(* Logix 5000 project; controller P5 vendor 1 type 14 code 92 rev 20.55; software revision 20.01 *)

TASK MainTask (continuous, watchdog 500 ms) : MainProgram

MODULES
   Local : vendor 1 type 14 code 92 (ICP 0, rev 20.55)
      P5_EN2T_PCN : 1756-EN2T (ICP 1, Ethernet 192.168.1.50, rev 10.1)
         P4 : 1756-EN2T (Ethernet 192.168.1.40, rev 10.1, Output RPI 10 ms)
            P4_CONTROLLER : vendor 1 type 14 code 92 (ICP 0, rev 20.1)
      P5_EN2TR_RIO : vendor 1 type 12 code 200 (ICP 2, Ethernet 192.168.0.40, rev 10.1)
         VSD501 : PowerFlex 525-EENET (Ethernet 192.168.0.57, rev 2.2, Output RPI 20 ms)
         VSD502 : PowerFlex 525-EENET (Ethernet 192.168.0.59, rev 3.1, Output RPI 20 ms)
         RIO5 : 1794-AENTR (Ethernet 192.168.0.52, rev 1.1, Output RPI 20 ms)
            RIO5_DI : 1794-IB32 (Flex 0, rev 1.1, Input RPI 20 ms)
            RIO5_DO : vendor 1 type 7 code 35 (Flex 1, rev 1.1)
            RIO5_AI : 1794-IE12 (Flex 2, rev 1.1, Output RPI 78 ms)
         WRIO5 : vendor 309 type 12 code 1000 (Ethernet 192.168.0.55, rev 3.1, Output RPI 20 ms)
            WRIO5_AI2 : 1734-IE4C (PointIO 2, rev 3.1, Input RPI 80 ms)
            WRIO5_AI1 : vendor 1 type 115 code 210 (PointIO 1, rev 3.1, Input RPI 80 ms)
END_MODULES

TYPE AIN_UDT :
STRUCT
   Pv : REAL;
   Heu : REAL;
   Leu : REAL;
   SAHH : REAL;
   SAH : REAL;
   SAL : REAL;
   SALL : REAL;
   AHH : BOOL;
   AH : BOOL;
   AL : BOOL;
   ALL : BOOL;
   Wifi_Enb : BOOL;
   Hty : BOOL;
   Sim : BOOL;
   Sim_PV : REAL;
END_STRUCT
END_TYPE

TYPE AUTOINP_UDT :
STRUCT
   ON : BOOL;
END_STRUCT
END_TYPE

TYPE ControllerLEDStatus :
STRUCT
   Off : BOOL;
   SolidGreen : BOOL;
   FlashingGreen : BOOL;
   SolidYellow : BOOL;
   FlashingYellow : BOOL;
   FlashingRed : BOOL;
   SolidRed : BOOL;
END_STRUCT
END_TYPE

TYPE DOSING_SETPOINT_UDT :
STRUCT
   High_Setpoint : REAL;
   Low_Setpoint : REAL;
END_STRUCT
END_TYPE

TYPE Duty2_UDT :
STRUCT
   Selection : INT;
   Pump_Running : BOOL;
   Selected_Pmp_Not_Avl : BOOL;
   Both_Pmp_Not_Avl : BOOL;
END_STRUCT
END_TYPE

TYPE FaultRecord :
STRUCT
   timelow : DINT;
   timehigh : DINT;
   type : INT;
   code : INT;
   info : DINT[8];
END_STRUCT
END_TYPE

TYPE FIT_UDT :
STRUCT
   Pv : REAL;
   Heu : REAL;
   Leu : REAL;
   SAHH : REAL;
   SAH : REAL;
   SAL : REAL;
   SALL : REAL;
   Totaliser : REAL;
   AHH : BOOL;
   AH : BOOL;
   AL : BOOL;
   ALL : BOOL;
   Sim : BOOL;
   Sim_PV : REAL;
   Wifi_Enb : BOOL;
   Rst_Totaliser : BOOL;
   Hty : BOOL;
END_STRUCT
END_TYPE

TYPE Logix_Status_FP :
STRUCT
   ClearMinorFaults : DINT;
   Sts_MinorFaultEvents : DINT;
   Sts_MinorFaultBits : DINT;
   Sts_Redundant : DINT;
   Set_FaceplateAnimation : DINT;
   Val_ProductCode : DINT;
   MemoryTemp : INT[29];
   Val_raw_data : INT;
   Sts_IO_LED_raw : INT;
   Sts_ProductCode : INT;
   Val_Force_data_raw : INT;
   MemoryRequestData : SINT[12];
   Sts_Force_Installed : BOOL;
   Sts_Force_Enabled : BOOL;
   Sts_Faulted : BOOL;
   Sts_Run : BOOL;
   Sts_Program : BOOL;
   Sts_Minor_fault : BOOL;
   Sts_Major_fault : BOOL;
   Sts_KS_in_run : BOOL;
   Sts_KS_in_program : BOOL;
   Sts_KS_in_remote : BOOL;
   Sts_Changingmodes : BOOL;
   Sts_Test : BOOL;
   Sts_Ladder_Working : BOOL;
   Cmd_ClearFaultRecord : BOOL;
   Set_Controller_Description : STRING;
   UpdateDelayTimer : TIMER;
   Val_MajorFault : FaultRecord;
   Val_MFS : FaultRecord;
   Sts_IO_LED : ControllerLEDStatus;
   Sts_Battery_LED : ControllerLEDStatus;
   MemoryData : Memory_Data;
   TEST : DINT;
END_STRUCT
END_TYPE

TYPE Memory_Data :
STRUCT
   Free_Mem_IO : DINT;
   Free_Mem_DT : DINT;
   Free_Memory : DINT;
   Total_Mem_IO : DINT;
   Total_Mem_DT : DINT;
   Total_Memory : DINT;
   Biggest_IO_Mem_Size_Ava : DINT;
   Biggest_DT_Mem_Size_Ava : DINT;
END_STRUCT
END_TYPE

TYPE MV_UDT :
STRUCT
   Cmd : INT;
   Status : INT;
   Reset : BOOL;
   Auto : BOOL;
   FTO : BOOL;
   FTC : BOOL;
   Avl : BOOL;
END_STRUCT
END_TYPE

TYPE PLANT_AUTO_UDT :
STRUCT
   ON : BOOL;
   OFF : BOOL;
END_STRUCT
END_TYPE

TYPE PLANT_UDT :
STRUCT
   START : BOOL;
   STOP : BOOL;
END_STRUCT
END_TYPE

TYPE PMP_UDT :
STRUCT
   Cmd : INT;
   Status : INT;
   RunMin : REAL;
   Total_RunMin : REAL;
   RunHr : REAL;
   Total_RunHr : REAL;
   Remote : BOOL;
   Auto : BOOL;
   Fault : BOOL;
   Avl : BOOL;
   Permissive : DINT;
   Shutdown : DINT;
   SD : DINT;
   Reset : BOOL;
   Reset_RunHr : BOOL;
   FTR : BOOL;
   FTS : BOOL;
END_STRUCT
END_TYPE

TYPE PRECONDITION_UDT :
STRUCT
   PERMISSIVE1 : BOOL;
   PERMISSIVE2 : BOOL;
   PERMISSIVE3 : BOOL;
   PERMISSIVE4 : BOOL;
   PERMISSIVE5 : BOOL;
   SHUTDOWN1 : BOOL;
   SHUTDOWN2 : BOOL;
   SHUTDOWN3 : BOOL;
   SHUTDOWN4 : BOOL;
   SHUTDOWN5 : BOOL;
END_STRUCT
END_TYPE

TYPE RED_STAT :
STRUCT
   Redundancy_status_of_the_controller : INT;
   Redundancy_state_of_the_partner : INT;
END_STRUCT
END_TYPE

TYPE SWITCH_UDT :
STRUCT
   Alarm : BOOL;
   Delay : DINT;
END_STRUCT
END_TYPE

TYPE UV_UDT :
STRUCT
   Cmd : INT;
   Status : INT;
   RunMin : REAL;
   Total_RunMin : REAL;
   RunHr : REAL;
   Total_RunHr : REAL;
   Remote : BOOL;
   Auto : BOOL;
   Fault : BOOL;
   Avl : BOOL;
   Permissive : DINT;
   Shutdown : DINT;
   SD : DINT;
   Reset : BOOL;
   Reset_RunHr : BOOL;
   FTR : BOOL;
   FTS : BOOL;
END_STRUCT
END_TYPE

TYPE VSD_UDT :
STRUCT
   Cmd : INT;
   Status : INT;
   RunMin : REAL;
   Total_RunMin : REAL;
   RunHr : REAL;
   Total_RunHr : REAL;
   Remote : BOOL;
   Auto : BOOL;
   Fault : BOOL;
   Avl : BOOL;
   Drive_Ready : BOOL;
   Speed : REAL;
   Speed_Command : REAL;
   Permissive : DINT;
   Shutdown : DINT;
   SD : DINT;
   Reset : BOOL;
   Reset_RunHr : BOOL;
   FTR : BOOL;
   FTS : BOOL;
END_STRUCT
END_TYPE

TYPE WIFI_UDT :
STRUCT
   PLC_WIFI : BOOL;
   RIO_WIFI : BOOL;
END_STRUCT
END_TYPE

ADD_ON_INSTRUCTION AIN_FBD   (* revision 1.0 *)
VAR_INPUT
   WRIO_Enb : BOOL; {visible}
   Raw_RIO : INT; {visible}
   Raw_WRIO : INT; {visible}
   L_Raw_RIO : INT; {visible}
   H_Raw_RIO : INT; {visible}
   L_Raw_WRIO : INT; {visible}
   H_Raw_WRIO : INT; {visible}
   HEU : INT; {visible}
   LEU : INT; {visible}
END_VAR
VAR_OUTPUT
   Hty : BOOL; {visible}
   Wifi_Enb : BOOL; {access Read Only, visible}
   AHH : BOOL; {visible}
   AH : BOOL; {access Read Only, visible}
   AL : BOOL; {access Read Only, visible}
   ALL : BOOL; {visible}
END_VAR
VAR_INPUT
   SAHH : REAL; {visible}
   SAH : REAL; {visible}
   SAL : REAL; {visible}
   SALL : REAL; {visible}
   Simulation : BOOL; {visible}
   RIO_Hty : BOOL; {visible}
   WRIO_Hty : BOOL; {visible}
END_VAR
VAR_IN_OUT
   Pv : REAL; {required}
   Sim_PV : REAL; {required}
   HMI : AIN_UDT; {required}
END_VAR
VAR
   SCALE : SCALE; {access None}
   ALM : ALARM; {access None}
   _Raw : INT; {access None}
   _L_Raw : INT; {access None}
   _H_Raw : INT; {access None}
   _Inst_Hty : BOOL; {access None}
END_VAR

ROUTINE Logic   (* structured text *)
   (*RIO and Wireless RIO Selection*)
   
   IF WRIO_Enb THEN
   	Wifi_Enb	:= 1;
   	_Raw		:= Raw_WRIO;
   	_H_Raw		:= H_Raw_WRIO;
   	_L_Raw		:= L_Raw_WRIO;
   	_Inst_Hty 	:= WRIO_Hty;
   ELSE
   	Wifi_Enb	:= 0;
   	_Raw		:= Raw_RIO;
   	_H_Raw		:= H_Raw_RIO;
   	_L_Raw		:= L_Raw_RIO;
   	_Inst_Hty 	:= RIO_Hty;
   END_IF;
   
   (*Calculation for PV*)
   IF Simulation THEN
   	Pv	:=Sim_PV;
   ELSE
   	SCALE.In		:=_Raw;
   	SCALE.InRawMax	:=_H_Raw;
   	SCALE.InRawMin	:=_L_Raw;
   	SCALE.InEUMax	:=HEU;
   	SCALE.InEUMin	:=LEU;
   	SCL(SCALE);
   
   	IF SCALE.Out<0 THEN
   		Pv	:= 0.0;
   	ELSE
   		Pv	:=SCALE.Out;
   	END_IF;
   
   	Sim_PV	:=Pv;
   
   END_IF;
   
   (*Alarms*)
   ALM.In			:=Pv;
   ALM.HHLimit		:=SAHH;
   ALM.HLimit		:=SAH;
   ALM.LLimit		:=SAL;
   ALM.LLLimit		:=SALL;
   ALM(ALM);
   
   AHH				:=ALM.HHAlarm;
   AH				:=ALM.HAlarm;
   AL				:=ALM.LAlarm;
   ALL				:=ALM.LLAlarm;
   
   Hty:= _Inst_Hty AND (_Raw > _L_Raw) AND (_Raw < _H_Raw)  ;
   
   
   
   
   
   
END_ROUTINE
END_ADD_ON_INSTRUCTION

ADD_ON_INSTRUCTION Duty2_FBD   (* revision 1.0 *)
VAR_INPUT
   AutoInp : BOOL; {visible}
   Selection : INT; {visible}
END_VAR
VAR_OUTPUT
   Start_Pmp1 : BOOL; {visible}
   Start_Pmp2 : BOOL; {visible}
END_VAR
VAR_IN_OUT
   PMP1 : VSD_UDT; {required}
   PMP2 : VSD_UDT; {required}
   HMI : Duty2_UDT; {required}
END_VAR

ROUTINE Logic   (* structured text *)
   IF PMP1.Status=2 OR PMP2.Status=2 THEN
   	HMI.Pump_Running := 1;
   ELSE
   	HMI.Pump_Running := 0;
   END_IF;
   
   HMI.Both_Pmp_Not_Avl		:= NOT PMP1.Avl AND NOT PMP2.Avl;
   
   IF AutoInp THEN
   	CASE Selection OF
   		(*PUMP 1 *)
   		1:
   			IF PMP1.Avl THEN
   				Start_Pmp1					:=1;
   				Start_Pmp2					:=0;
   				HMI.Selected_Pmp_Not_Avl	:=0;
   			ELSIF NOT PMP1.Avl AND PMP2.Avl THEN
   				Start_Pmp1					:=0;
   				Start_Pmp2					:=1;
   				HMI.Selected_Pmp_Not_Avl	:=1;
   			ELSIF NOT PMP1.Avl AND NOT PMP2.Avl	THEN
   				Start_Pmp1					:=0;
   				Start_Pmp2					:=0;
   			ELSE
   				HMI.Selected_Pmp_Not_Avl	:=0;
   			END_IF;
   
   		(*PUMP 2 *)
   		2:
   			IF PMP2.Avl THEN
   				Start_Pmp1					:=0;
   				Start_Pmp2					:=1;
   				HMI.Selected_Pmp_Not_Avl	:=0;
   			ELSIF NOT PMP2.Avl AND PMP1.Avl THEN
   				Start_Pmp1					:=1;
   				Start_Pmp2					:=0;
   				HMI.Selected_Pmp_Not_Avl	:=1;
   			ELSIF NOT PMP1.Avl AND NOT PMP2.Avl	THEN
   				Start_Pmp1					:=0;
   				Start_Pmp2					:=0;
   			ELSE
   				HMI.Selected_Pmp_Not_Avl	:=0;
   			END_IF;
   	END_CASE;
   ELSE
   	Start_Pmp1					:=0;
   	Start_Pmp2					:=0;
   END_IF;
   
   
END_ROUTINE
END_ADD_ON_INSTRUCTION

ADD_ON_INSTRUCTION FIT_FBD   (* revision 1.0 *)
VAR_INPUT
   WRIO_Enb : BOOL; {visible}
   Raw_RIO : INT; {visible}
   Raw_WRIO : INT; {visible}
   L_Raw_RIO : INT; {visible}
   H_Raw_RIO : INT; {visible}
   L_Raw_WRIO : INT; {visible}
   H_Raw_WRIO : INT; {visible}
   HEU : REAL; {visible}
   LEU : REAL; {visible}
END_VAR
VAR_OUTPUT
   Hty : BOOL; {visible}
   Wifi_Enb : BOOL; {visible}
   AHH : BOOL; {visible}
   AH : BOOL; {access Read Only, visible}
   AL : BOOL; {access Read Only, visible}
   ALL : BOOL; {visible}
END_VAR
VAR_INPUT
   SAHH : REAL; {visible}
   SAH : REAL; {visible}
   SAL : REAL; {visible}
   SALL : REAL; {visible}
   Simulation : BOOL; {visible}
   RIO_Hty : BOOL; {visible}
   WRIO_Hty : BOOL; {visible}
   Totaliser_Enb : BOOL; {visible}
   Rst_Totaliser : BOOL; {visible}
END_VAR
VAR_IN_OUT
   Totaliser : REAL; {required}
   Pv : REAL; {required}
   Sim_Pv : REAL; {required}
   HMI : FIT_UDT; {required}
END_VAR
VAR
   SCALE : SCALE; {access None}
   ALM : ALARM; {access None}
   TON : FBD_TIMER; {access None}
   _SEC_P : BOOL; {access None}
   _Inst_Hty : BOOL; {access None}
   _L_Raw : INT; {access None}
   _H_Raw : INT; {access None}
   _Raw : INT; {access None}
   R_TRIG : FBD_ONESHOT; {access None}
END_VAR

ROUTINE Logic   (* structured text *)
   (*RIO and Wireless RIO Selection*)
   
   IF WRIO_Enb THEN
   	Wifi_Enb	:= 1;
   	_Raw		:= Raw_WRIO;
   	_H_Raw		:= H_Raw_WRIO;
   	_L_Raw		:= L_Raw_WRIO;
   	_Inst_Hty 	:= WRIO_Hty;
   ELSE
   	Wifi_Enb	:= 0;
   	_Raw		:= Raw_RIO;
   	_H_Raw		:= H_Raw_RIO;
   	_L_Raw		:= L_Raw_RIO;
   	_Inst_Hty 	:= RIO_Hty;
   END_IF;
   
   (*Calculation for PV*)
   IF Simulation THEN
   	Pv	:= Sim_Pv   ;
   ELSE
   	SCALE.In		:=_Raw;
   	SCALE.InRawMax	:=_H_Raw;
   	SCALE.InRawMin	:=_L_Raw;
   	SCALE.InEUMax	:=HEU;
   	SCALE.InEUMin	:=LEU;
   	SCL(SCALE);
   	IF SCALE.Out>0 THEN
   		Pv	:=SCALE.Out;
   	ELSIF SCALE.Out<=0 THEN
   		Pv	:=0.0;
   	END_IF;
   
   	Sim_Pv	:=Pv;
   END_IF;
   
   (*Alarms*)
   ALM.In			:=Pv;
   ALM.HHLimit		:=SAHH;
   ALM.HLimit		:=SAH;
   ALM.LLimit		:=SAL;
   ALM.LLLimit		:=SALL;
   ALM(ALM);
   
   AHH				:=ALM.HHAlarm;
   AH				:=ALM.HAlarm;
   AL				:=ALM.LAlarm;
   ALL				:=ALM.LLAlarm;
   
   (*SECOND PULSE*)
   TON.PRE	:=1000;
   TON.TimerEnable	:=1;
   TONR(TON );
   R_TRIG.InputBit :=TON.DN ;
   OSRI( R_TRIG);
   _SEC_P  := R_TRIG.OutputBit;
   TON.Reset := _SEC_P;
   
   IF Totaliser_Enb THEN
   	IF _SEC_P THEN
   		HMI.Totaliser := HMI.Totaliser +  (ABS(Pv) / 3600 );
   	END_IF;
   END_IF;
   
   IF  Rst_Totaliser   THEN
   	HMI.Totaliser	:=0;
   END_IF;
   
   Hty:= _Inst_Hty AND (_Raw > _L_Raw) AND (_Raw < _H_Raw)  ;
   
   
   
   
   
   
END_ROUTINE
END_ADD_ON_INSTRUCTION

ADD_ON_INSTRUCTION MV_FBD   (* revision 1.0 *)
VAR_INPUT
   Auto : BOOL; {visible}
END_VAR
VAR_OUTPUT
   Cmd_Open : BOOL; {visible}
   Cmd_Close : BOOL; {visible}
   FTO : BOOL; {visible}
   FTC : BOOL; {access Read Only, visible}
END_VAR
VAR_INPUT
   AutoInp : BOOL; {visible}
   ZSO : BOOL; {visible}
   Open_TM : DINT; {visible}
   ZSC : BOOL; {visible}
   Close_TM : DINT; {visible}
END_VAR
VAR_IN_OUT
   Cmd : INT; {required}
   HMI : MV_UDT; {required}
END_VAR
VAR
   TON_Open_TM : FBD_TIMER; {access None}
   TON_Close_TM : FBD_TIMER; {access None}
END_VAR

ROUTINE Logic   (* structured text *)
   (*Fail to Close*)
   TON_Close_TM.PRE 			:= 	Close_TM*1000;
   TON_Close_TM.TimerEnable 	:=  Cmd_Close;
   TONR(TON_Close_TM);
   
   (*Fail to Open*)
   TON_Open_TM.PRE 			:= 	Open_TM*1000;
   TON_Open_TM.TimerEnable 	:= 	Cmd_Open;
   TONR(TON_Open_TM);
   
   IF ZSC THEN
   	HMI.Status	:=1;
   ELSIF ZSO THEN
   	HMI.Status	:=2;
   ELSE
   	HMI.Status	:=0;
   END_IF;
   
   HMI.Avl:= Auto AND NOT FTC AND NOT FTO;
   
   IF HMI.Reset THEN
   	(*IF NOT TON_Close_TM.DN AND ZSC THEN*)
   			FTC		:= 0;
   	(*END_IF;*)
   	(*IF NOT TON_Open_TM.DN AND ZSO THEN*)
   			FTO		:= 0;
   	(*END_IF;*)
   END_IF;
   
   IF  NOT Auto THEN
   	CASE HMI.Cmd OF
   		1:	(*CLOSE*)
   			Cmd_Close	:= 1;
   			Cmd_Open	:= 0;
   			IF TON_Close_TM.DN AND (NOT ZSC) THEN
   				FTC		:= 1;
   				FTO		:= 0;
   			END_IF;
   		2:	(*OPEN*)
   			IF FTO OR FTC    THEN
   				HMI.Cmd := 1;
   			END_IF;
   
   			IF NOT FTC AND NOT FTO THEN
   				Cmd_Close	:= 0;
   				Cmd_Open	:= 1;
   			END_IF;
   
   			IF TON_Open_TM.DN AND (NOT ZSO) THEN
   				FTC		:= 0;
   				FTO		:= 1;
   				HMI.Cmd := 1;
   			END_IF;
   	END_CASE;
   ELSE
   	(*Maintain Last status when switching from Auto to Manual*)
   	IF ZSO THEN
   		Cmd	:= 2;
   	END_IF;
   	IF ZSC THEN
   		Cmd	:= 1;
   	END_IF;
   
   	IF  AutoInp AND (NOT FTC AND NOT FTO) THEN
   		Cmd_Close	:= 0;
   		Cmd_Open	:= 1;
   		IF TON_Open_TM.DN AND (NOT ZSO) THEN
   			FTC		:= 0;
   			FTO		:= 1;
   		END_IF;
   	ELSE
   		Cmd_Close	:= 1;
   		Cmd_Open	:= 0;
   		IF TON_Close_TM.DN AND (NOT ZSC) THEN
   			FTC		:= 1;
   			FTO		:= 0;
   		END_IF;
   	END_IF;
   END_IF;
   
   
END_ROUTINE
END_ADD_ON_INSTRUCTION

ADD_ON_INSTRUCTION PMP_FBD   (* revision 1.0 *)
VAR_OUTPUT
   Cmd_Start : BOOL; {visible}
   Avl : BOOL; {visible}
   Fault : BOOL; {visible}
   FT_Stop : BOOL; {visible}
   FT_Start : BOOL; {visible}
   RunHr : REAL; {visible}
   Total_RunHr : REAL; {visible}
   SD : DINT; {access Read Only, visible}
END_VAR
VAR_INPUT
   Auto : BOOL; {visible}
   AutoInp : BOOL; {visible}
   Remote : BOOL; {visible}
   Run : BOOL; {visible}
   Trip : BOOL; {visible}
   Start_TM : DINT; {visible}
   Stop_TM : DINT; {visible}
   Rst : BOOL; {visible}
   Rst_RunHr : BOOL; {visible}
   Permissive : DINT; {visible}
   Shutdown : DINT; {visible}
END_VAR
VAR_IN_OUT
   RunMin : REAL; {required}
   Total_RunMin : REAL; {required}
   Cmd : INT; {required}
   HMI : PMP_UDT; {required}
END_VAR
VAR
   TON_Start_TM : FBD_TIMER; {access None}
   TON_Stop_TM : FBD_TIMER; {access None}
   _Min_P : BOOL; {access None}
   TON_Min : FBD_TIMER; {access None}
   R_TRIG_SEC : FBD_ONESHOT; {access None}
END_VAR

ROUTINE Logic   (* structured text *)
   (*Fail to Start*)
   TON_Start_TM.PRE 			:= 	Start_TM*1000;
   TON_Start_TM.TimerEnable 	:=  Cmd_Start;
   TONR(TON_Start_TM);
   
   (*Fail to Stop*)
   TON_Stop_TM.PRE 			:= 	Stop_TM*1000;
   TON_Stop_TM.TimerEnable 	:=  NOT Cmd_Start;
   TONR(TON_Stop_TM);
   
   IF (NOT Run) THEN
   	HMI.Status	:=1;
   ELSE
   	HMI.Status	:=2;
   END_IF;
   
   IF Fault THEN
   	HMI.Fault:= 1;
   ELSE
   	HMI.Fault:= 0;
   END_IF;
   
   IF HMI.Reset THEN
   	IF NOT TON_Stop_TM.DN THEN
   			FT_Stop		:= 0;
   	END_IF;
   	IF NOT TON_Start_TM.DN THEN
   			FT_Start	:= 0;
   	END_IF;
   
   	SD :=0;
   
   END_IF;
   
   Fault		:=Trip OR SD<>0;
   HMI.Remote	:=Remote;
   Avl:= Auto AND Remote AND NOT Fault AND NOT FT_Start AND NOT FT_Stop AND SD=0 ;
   
   IF Remote THEN
   	IF  NOT Auto THEN
   		CASE HMI.Cmd OF
   			1:	(*Stop*)
   				Cmd_Start	:=0;
   				IF TON_Stop_TM.DN AND Run THEN
   					FT_Start	:= 0;
   					FT_Stop		:= 1;
   				END_IF;
   			2:	(*OPEN*)
   				IF NOT Fault AND NOT FT_Start AND NOT FT_Stop AND (Permissive=-1) AND HMI.SD=0 THEN
   					Cmd_Start	:= 1;
   				ELSIF Cmd_Start AND (HMI.SD<>0) OR Fault THEN
   					SD				:= HMI.SD;
   					Cmd_Start		:= 0;
   					HMI.Cmd 		:= 1;
   				ELSIF (Permissive<>-1) THEN
   					HMI.Cmd 		:= 1;
   				END_IF;
   
   				IF TON_Start_TM.DN AND NOT Run THEN
   					FT_Start	:= 1;
   					FT_Stop		:= 0;
   					Cmd_Start	:= 0;
   					HMI.Cmd 	:= 1;
   				END_IF;
   		END_CASE;
   	ELSE
   		IF Run THEN
   			Cmd	:= 2;
   		END_IF;
   		IF (NOT Run) OR Fault OR FT_Start OR FT_Stop THEN
   			Cmd	:= 1;
   		END_IF;
   
   		IF  AutoInp  THEN
   			IF NOT Fault AND NOT FT_Start AND NOT FT_Stop AND (Permissive=-1) AND HMI.SD=0  THEN
   				Cmd_Start	:=1;
   			ELSIF Cmd_Start OR (HMI.SD<>0) OR Fault THEN
   				SD			:= HMI.SD;
   				Cmd_Start	:=0;
   			END_IF;
   
   			IF TON_Start_TM.DN AND NOT Run THEN
   				FT_Start	:= 1;
   				FT_Stop		:= 0;
   				Cmd_Start	:= 0;
   				HMI.Cmd 	:= 1;
   			END_IF;
   		ELSE
   			Cmd_Start	:=0;
   			IF TON_Stop_TM.DN AND Run THEN
   				FT_Start	:= 0;
   				FT_Stop		:= 1;
   
   			END_IF;
   		END_IF;
   	END_IF;
   
   ELSE (*Local*)
   	Cmd_Start	:=0;
   	Cmd	:= 1;
   
   	FT_Start	:= 0;
   	FT_Stop		:= 0;
   
   
   
   
   	(*	IF Run THEN
   			Cmd	:= 2;
   		END_IF;
   		IF (NOT Run) OR Fault OR FT_Start OR FT_Stop THEN
   			Cmd	:= 1;
   		END_IF;
   		*)
   END_IF;
   
   (*1 MIN PULSE*)
   TON_Min.PRE	:=60000;
   TON_Min.TimerEnable	:=1;
   TONR(TON_Min );
   R_TRIG_SEC.InputBit :=TON_Min.DN ;
   OSRI( R_TRIG_SEC);
   _Min_P  := R_TRIG_SEC.OutputBit;
   TON_Min.Reset 	:= _Min_P;
   
   IF Run THEN
   	IF _Min_P THEN
   		RunMin 			:=RunMin + 1.0;
   		Total_RunMin	:=Total_RunMin + 1.0;
   	END_IF;
   END_IF;
   
   RunHr 				:=RunMin/60.0;
   Total_RunHr			:=Total_RunMin/60.0;
   
   IF  Rst_RunHr THEN
   	RunMin	:=0;
   END_IF;
   
   
   
END_ROUTINE
END_ADD_ON_INSTRUCTION

ADD_ON_INSTRUCTION SWITCH_FBD   (* revision 1.0 *)
VAR_INPUT
   Alarm : BOOL; {visible}
   Delay : DINT; {required}
END_VAR
VAR_OUTPUT
   Status : BOOL; {access None, required}
END_VAR
VAR_IN_OUT
   HMI : SWITCH_UDT; {required}
END_VAR
VAR
   TON_Delay_Sec : FBD_TIMER; {access None}
END_VAR

ROUTINE Logic   (* structured text *)
   (*Delay for Alarm*)
   TON_Delay_Sec.PRE 			:= 	Delay*1000;
   TON_Delay_Sec.TimerEnable 	:=  Alarm;
   TONR(TON_Delay_Sec);
   
   Status := TON_Delay_Sec.DN ;
END_ROUTINE
END_ADD_ON_INSTRUCTION

ADD_ON_INSTRUCTION UV_FBD   (* revision 1.0 *)
VAR_OUTPUT
   Cmd_Start : BOOL; {visible}
   Avl : BOOL; {visible}
   Fault : BOOL; {visible}
   FT_Stop : BOOL; {visible}
   FT_Start : BOOL; {visible}
   RunHr : REAL; {visible}
   Total_RunHr : REAL; {visible}
END_VAR
VAR_INPUT
   Auto : BOOL; {visible}
   AutoInp : BOOL; {visible}
   Remote : BOOL; {visible}
   Run : BOOL; {visible}
   Trip : BOOL; {visible}
   Start_TM : DINT; {visible}
   Stop_TM : DINT; {visible}
   Rst : BOOL; {visible}
   Rst_RunHr : BOOL; {visible}
   Permissive : INT; {visible}
   Shutdown : INT; {visible}
END_VAR
VAR_IN_OUT
   RunMin : REAL; {required}
   Total_RunMin : REAL; {required}
   Cmd : INT; {required}
   HMI : UV_UDT; {required}
END_VAR
VAR
   TON_Start_TM : FBD_TIMER; {access None}
   TON_Stop_TM : FBD_TIMER; {access None}
   _Min_P : BOOL; {access None}
   TON_Min : FBD_TIMER; {access None}
   R_TRIG_SEC : FBD_ONESHOT; {access None}
END_VAR

ROUTINE Logic   (* structured text *)
   (*Fail to Start*)
   TON_Start_TM.PRE 			:= 	Start_TM*1000;
   TON_Start_TM.TimerEnable 	:=  Cmd_Start;
   TONR(TON_Start_TM);
   
   (*Fail to Stop*)
   TON_Stop_TM.PRE 			:= 	Stop_TM*1000;
   TON_Stop_TM.TimerEnable 	:=  NOT Cmd_Start;
   TONR(TON_Stop_TM);
   
   IF (NOT Run) THEN
   	HMI.Status	:=1;
   ELSE
   	HMI.Status	:=2;
   END_IF;
   
   IF Fault THEN
   	HMI.Fault:= 1;
   ELSE
   	HMI.Fault:= 0;
   END_IF;
   
   IF HMI.Reset THEN
   	IF NOT TON_Stop_TM.DN THEN
   			FT_Stop		:= 0;
   	END_IF;
   	IF NOT TON_Start_TM.DN THEN
   			FT_Start	:= 0;
   	END_IF;
   END_IF;
   
   
   HMI.Remote	:=Remote;
   Avl:= Auto AND Remote AND NOT Fault AND NOT FT_Stop AND NOT FT_Stop   ;
   
   
   
   IF Remote THEN
   	IF  NOT Auto THEN
   		CASE HMI.Cmd OF
   			1:	(*Stop*)
   				Cmd_Start	:=0;
   				IF TON_Stop_TM.DN AND Run THEN
   					FT_Start	:= 0;
   					FT_Stop		:= 1;
   				END_IF;
   			2:	(*OPEN*)
   				IF NOT Fault AND (NOT FT_Start OR FT_Stop) AND (Permissive=-1) THEN
   					Cmd_Start	:= 1;
   				END_IF;
   
   				IF (Shutdown<>0) OR Fault THEN
   					Cmd_Start	:= 0;
   					HMI.Cmd 	:= 1;
   				END_IF;
   
   				IF TON_Start_TM.DN AND NOT Run THEN
   					FT_Start	:= 1;
   					FT_Stop		:= 0;
   					Cmd_Start	:= 0;
   					HMI.Cmd 	:= 1;
   				END_IF;
   		END_CASE;
   	ELSE
   		IF Run THEN
   			Cmd	:= 2;
   		END_IF;
   		IF (NOT Run) OR Fault OR FT_Start OR FT_Stop THEN
   			Cmd	:= 1;
   		END_IF;
   
   		IF  AutoInp  THEN
   			IF NOT Fault AND (NOT FT_Start OR FT_Stop) AND (Permissive=-1) THEN
   				Cmd_Start	:=1;
   			END_IF;
   
   			IF (Shutdown<>0) OR Fault THEN
   				Cmd_Start	:=0;
   			END_IF;
   
   			IF TON_Start_TM.DN AND NOT Run THEN
   				FT_Start	:= 1;
   				FT_Stop		:= 0;
   				Cmd_Start	:= 0;
   				HMI.Cmd 	:= 1;
   			END_IF;
   		ELSE
   			Cmd_Start	:=0;
   			IF TON_Stop_TM.DN AND Run THEN
   				FT_Start	:= 0;
   				FT_Stop		:= 1;
   
   			END_IF;
   		END_IF;
   	END_IF;
   
   ELSE (*Local*)
   	Cmd_Start	:=0;
   	Cmd	:= 1;
   
   	(*	IF Run THEN
   			Cmd	:= 2;
   		END_IF;
   		IF (NOT Run) OR Fault OR FT_Start OR FT_Stop THEN
   			Cmd	:= 1;
   		END_IF;
   		*)
   END_IF;
   
   (*1 MIN PULSE*)
   TON_Min.PRE	:=60000;
   TON_Min.TimerEnable	:=1;
   TONR(TON_Min );
   R_TRIG_SEC.InputBit :=TON_Min.DN ;
   OSRI( R_TRIG_SEC);
   _Min_P  := R_TRIG_SEC.OutputBit;
   TON_Min.Reset 	:= _Min_P;
   
   IF Run THEN
   	IF _Min_P THEN
   		RunMin 			:=RunMin + 1.0;
   		Total_RunMin	:=Total_RunMin + 1.0;
   	END_IF;
   END_IF;
   
   RunHr 				:=RunMin/60.0;
   Total_RunHr			:=Total_RunMin/60.0;
   
   IF  Rst_RunHr THEN
   	RunMin	:=0;
   END_IF;
   
   
   
END_ROUTINE
END_ADD_ON_INSTRUCTION

ADD_ON_INSTRUCTION VSD_FBD   (* revision 1.0 *)
VAR_OUTPUT
   Avl : BOOL; {visible}
   Fault : BOOL; {visible}
   FT_Stop : BOOL; {visible}
   FT_Start : BOOL; {visible}
   RunHr : REAL; {visible}
   Total_RunHr : REAL; {visible}
   Speed : REAL; {visible}
   Rdy : BOOL; {visible}
   SD : DINT; {access Read Only, visible}
END_VAR
VAR_INPUT
   Auto : BOOL; {visible}
   AutoInp : BOOL; {visible}
   Remote : BOOL; {visible}
   Run : BOOL; {visible}
   Trip : BOOL; {visible}
   Start_PB : BOOL; {visible}
   Start_TM : DINT; {visible}
   Stop_TM : DINT; {visible}
   Rst : BOOL; {visible}
   Rst_RunHr : BOOL; {visible}
   AutoSpeed : REAL; {visible}
   Speed_Cmd : REAL; {visible}
   Permissive : DINT; {visible}
   Shutdown : DINT; {visible}
END_VAR
VAR_IN_OUT
   VSD_In : AB:PowerFlex525V_EENET_Drive:I:0; {required}
   VSD_Out : AB:PowerFlex525V_EENET_Drive:O:0; {required}
   RunMin : REAL; {required}
   Total_RunMin : REAL; {required}
   Cmd : INT; {required}
   HMI : VSD_UDT; {required}
END_VAR
VAR
   TON_Start_TM : FBD_TIMER; {access None}
   TON_Stop_TM : FBD_TIMER; {access None}
   _Min_P : BOOL; {access None}
   TON_Min : FBD_TIMER; {access None}
   R_TRIG_SEC : FBD_ONESHOT; {access None}
END_VAR

ROUTINE Logic   (* structured text *)
   (*Fail to Start*)
   TON_Start_TM.PRE 			:= 	Start_TM*1000;
   TON_Start_TM.TimerEnable 	:=  VSD_Out.Start;
   TONR(TON_Start_TM);
   
   (*Fail to Stop*)
   TON_Stop_TM.PRE 			:= 	Stop_TM*1000;
   TON_Stop_TM.TimerEnable 	:=  VSD_Out.Stop;
   TONR(TON_Stop_TM);
   
   IF (NOT VSD_In.Active) THEN
   	HMI.Status	:=1;
   ELSE
   	HMI.Status	:=2;
   END_IF;
   
   Rdy				:= VSD_In.Ready;
   Speed			:= VSD_In.OutputFreq/100;
   HMI.Remote		:= Remote;
   
   Avl:= Auto AND Remote AND NOT Fault AND NOT FT_Start AND NOT FT_Stop AND SD=0;  ;
   HMI.Fault:= VSD_In.Faulted OR Trip OR SD<>0;
   
   
   
   IF HMI.Reset THEN
   	VSD_Out.ClearFaults:=1;
   	HMI.SHUTDOWN:=0;
   
   	IF NOT TON_Stop_TM.DN THEN
   			FT_Stop		:= 0;
   	END_IF;
   	IF NOT TON_Start_TM.DN THEN
   			FT_Start	:= 0;
   	END_IF;
   
   	SD:=0;
   END_IF;
   
   IF Remote THEN
   	IF  NOT Auto THEN
   		CASE HMI.Cmd OF
   			1:	(*Stop*)
   
   				VSD_Out.Start		:=0;
   				VSD_Out.Stop		:=1;
   				VSD_Out.FreqCommand	:=Speed_Cmd;
   
   				IF TON_Stop_TM.DN AND VSD_In.Active THEN
   					FT_Start	:= 0;
   					FT_Stop		:= 1;
   				END_IF;
   			2:	(*Start*)
   				IF NOT VSD_In.Faulted AND (NOT FT_Start OR FT_Stop) AND (Permissive=-1) AND HMI.SD=0 THEN
   					VSD_Out.Start		:=1;
   					VSD_Out.Stop		:=0;
   			        VSD_Out.FreqCommand	:=Speed_Cmd*100;
   
   				ELSIF VSD_Out.Start OR (HMI.SD<>0) OR Fault THEN
   					SD 					:=HMI.SD;
   					VSD_Out.Start		:=0;
   					VSD_Out.Stop		:=1;
   					VSD_Out.FreqCommand	:=Speed_Cmd*100;
   					HMI.Cmd 	:= 1;
   				ELSIF (Permissive<>-1) THEN
   					HMI.Cmd 		:= 1;
   				END_IF;
   
   				IF TON_Start_TM.DN AND NOT Run THEN
   					FT_Start		:=1;
   					FT_Stop			:=0;
   					VSD_Out.Start	:=0;
   					VSD_Out.Stop	:=1;
   					HMI.Cmd 		:=1;
   				END_IF;
   		END_CASE;
   	ELSE
   		IF VSD_In.Active THEN
   			Cmd	:= 2;
   		END_IF;
   		IF (NOT VSD_In.Active) OR VSD_In.Faulted OR FT_Start OR FT_Stop THEN
   			Cmd	:= 1;
   		END_IF;
   
   		IF  AutoInp  THEN
   			IF NOT VSD_In.Faulted AND (NOT FT_Start OR FT_Stop) AND (Permissive=-1) AND HMI.SD=0 THEN
   				VSD_Out.Start		:=1;
   				VSD_Out.Stop		:=0;
   				VSD_Out.FreqCommand	:=AutoSpeed*100;
   
   			ELSIF VSD_Out.Start OR (HMI.SD<>0) OR Fault THEN
   				SD 					:=HMI.SD;
   				VSD_Out.Start		:=0;
   				VSD_Out.Stop		:=1;
   				VSD_Out.FreqCommand	:=AutoSpeed*100;
   				HMI.Cmd 			:= 1;
   			END_IF;
   
   			IF TON_Start_TM.DN AND NOT VSD_In.Active THEN
   				VSD_Out.Start		:=0;
   				VSD_Out.Stop		:=1;
   				VSD_Out.FreqCommand	:=AutoSpeed*100;
   				HMI.Cmd 			:= 1;
   			END_IF;
   		ELSE
   				VSD_Out.Start		:=0;
   				VSD_Out.Stop		:=1;
   			IF TON_Stop_TM.DN AND VSD_In.Active THEN
   				FT_Start	:= 0;
   				FT_Stop		:= 1;
   
   			END_IF;
   		END_IF;
   	END_IF;
   
   ELSE (*Local*)
   		IF Start_PB THEN
   			VSD_Out.Start 	:=1;
   			VSD_Out.Stop	:=0;
   				(*	VSD_Out.FreqCommand	:=Speed_Cmd*100; *)
   				 VSD_Out.FreqCommand	:=Speed_Cmd*110;
   		ELSE
   			VSD_Out.Start 	:=0;
   			VSD_Out.Stop	:=1;
   				(*	VSD_Out.FreqCommand	:=Speed_Cmd*100; *)
   				 VSD_Out.FreqCommand	:=Speed_Cmd*110;
   		END_IF;
   
   
   		IF Run THEN
   			Cmd	:= 2;
   		END_IF;
   		IF (NOT Run) OR Fault OR FT_Start OR FT_Stop THEN
   			Cmd	:= 1;
   		END_IF;
   END_IF;
   
   (*1 MIN PULSE*)
   TON_Min.PRE	:=60000;
   TON_Min.TimerEnable	:=1;
   TONR(TON_Min );
   R_TRIG_SEC.InputBit :=TON_Min.DN ;
   OSRI( R_TRIG_SEC);
   _Min_P  := R_TRIG_SEC.OutputBit;
   TON_Min.Reset 	:= _Min_P;
   
   IF Run OR VSD_In.Active THEN
   	IF _Min_P THEN
   		RunMin :=RunMin + 1.0;
   		Total_RunMin	:=Total_RunMin + 1.0;
   	END_IF;
   END_IF;
   
   RunHr 				:=RunMin/60.0;
   Total_RunHr			:=Total_RunMin/60.0;
   
   IF  Rst_RunHr THEN
   	RunMin	:=0;
   END_IF;
   
   
   
END_ROUTINE
END_ADD_ON_INSTRUCTION

VAR_GLOBAL   (* controller tags *)
   _FIT501_Tot_Enb : BOOL;
   _FIT502_Tot_Enb : BOOL;
   _FIT503_Tot_Enb : BOOL := 1;
   _FIT504_Tot_Enb : BOOL := 1;
   _MIN_P : BOOL;
   _MV501_AutoInp : BOOL;
   _MV502_AutoInp : BOOL;
   _MV503_AutoInp : BOOL;
   _MV504_AutoInp : BOOL;
   _NEXT : BOOL;
   _P401_AutoInp : BOOL;
   _P402_AutoInp : BOOL;
   _P403_AutoInp : BOOL;
   _P404_AutoInp : BOOL;
   _P501_AutoInp : BOOL;
   _P501_AutoSpeed : REAL;
   _P502_AutoInp : BOOL;
   _P502_AutoSpeed : REAL;
   _P50X_AutoSpeed : REAL := 10.0;
   _P_NAHSO3_ORP_DUTY_AutoInp : BOOL;
   _P_NAHSO3_ORP_DUTY_SR : DOMINANT_SET := (Reset := 1, OutNot := 1);
   _P_RO_FEED_DUTY_AutoInp : BOOL;
   _P_RO_FEED_DUTY_SR : DOMINANT_SET := (Set := 1, Out := 1);
   _P_RO_HIGH_AutoInp : BOOL;
   _P_UF_FEED_DUTY_AutoInp : BOOL := 1;
   _SEC_P : BOOL;
   _SEC_P1 : BOOL;
   _SEC_TEST : INT := -6124;
   _SEC_TEST1 : INT := 2391;
   _STOP : BOOL;
   _UV401_AutoInp : BOOL := 1;
   _UV_SR : DOMINANT_SET := (Set := 1, Out := 1);
   AI_AIT_401_HRDNSS : INT := -11;
   AI_AIT_401_HRDNSS_HTY : BOOL := 1;
   AI_AIT_402_ORP : INT := -17;
   AI_AIT_402_ORP_HTY : BOOL := 1;
   AI_AIT_501_PH : INT := 18894;
   AI_AIT_501_PH_HTY : BOOL := 1;
   AI_AIT_502_ORP : INT := 9002;
   AI_AIT_502_ORP_HTY : BOOL := 1;
   AI_AIT_503_COND : INT := 5384;
   AI_AIT_503_COND_HTY : BOOL := 1;
   AI_AIT_504_COND : INT := 933;
   AI_AIT_504_COND_HTY : BOOL := 1;
   AI_FIT_401_FLOW : INT := -19;
   AI_FIT_401_FLOW_HTY : BOOL := 1;
   AI_FIT_501_FLOW : INT := 15;
   AI_FIT_501_FLOW_HTY : BOOL := 1;
   AI_FIT_502_FLOW : INT := -9;
   AI_FIT_502_FLOW_HTY : BOOL := 1;
   AI_FIT_503_FLOW : INT := -24;
   AI_FIT_503_FLOW_HTY : BOOL := 1;
   AI_FIT_504_FLOW : INT := -26;
   AI_FIT_504_FLOW_HTY : BOOL := 1;
   AI_LIT_401_LEVEL : INT := -9;
   AI_LIT_401_LEVEL_HTY : BOOL := 1;
   AI_PIT_501_PRESS : INT := 722;
   AI_PIT_501_PRESS_HTY : BOOL := 1;
   AI_PIT_502_PRESS : INT := -21;
   AI_PIT_502_PRESS_HTY : BOOL := 1;
   AI_PIT_503_PRESS : INT := 402;
   AI_PIT_503_PRESS_HTY : BOOL := 1;
   AI_RIO4_SPARE_03 : INT;
   AI_RIO4_SPARE_03_HTY : BOOL;
   AI_RIO4_SPARE_04 : INT;
   AI_RIO4_SPARE_04_HTY : BOOL;
   AI_RIO4_SPARE_05 : INT;
   AI_RIO4_SPARE_05_HTY : BOOL;
   AI_RIO4_SPARE_06 : INT;
   AI_RIO4_SPARE_06_HTY : BOOL;
   AI_RIO4_SPARE_07 : INT;
   AI_RIO4_SPARE_07_HTY : BOOL;
   AI_RIO4_SPARE_08 : INT;
   AI_RIO4_SPARE_08_HTY : BOOL;
   AI_RIO4_SPARE_09 : INT;
   AI_RIO4_SPARE_09_HTY : BOOL;
   AI_RIO4_SPARE_10 : INT;
   AI_RIO4_SPARE_10_HTY : BOOL;
   AI_RIO4_SPARE_11 : INT;
   AI_RIO4_SPARE_11_HTY : BOOL := 1;
   AI_RIO5_SPARE_11 : INT := -7703;
   AIT401_FB : AIN_FBD := (Raw_RIO := -11, Raw_WRIO := 3266, H_Raw_RIO := 31208, L_Raw_WRIO := 3277, H_Raw_WRIO := 16383, HEU := 2, Hty := 1, AL := 1, ALL := 1, RIO_Hty := 1);
   AIT401_FB_01 : AIN_FBD;
   AIT402_FB : AIN_FBD := (Raw_RIO := -17, Raw_WRIO := 3268, H_Raw_RIO := 31208, L_Raw_WRIO := 3277, H_Raw_WRIO := 16383, HEU := 2, Hty := 1, AL := 1, ALL := 1, RIO_Hty := 1);
   AIT501_FB : AIN_FBD := (Raw_RIO := 18889, Raw_WRIO := 10247, H_Raw_RIO := 31208, L_Raw_WRIO := 3277, H_Raw_WRIO := 16383, HEU := 12, LEU := 2, Hty := 1, AHH := 1, AH := 1, RIO_Hty := 1);
   AIT502_FB : AIN_FBD := (Raw_RIO := 9002, Raw_WRIO := 6637, H_Raw_RIO := 31208, L_Raw_WRIO := 3277, H_Raw_WRIO := 16383, HEU := 800, Hty := 1, SAHH := 300.0, SAH := 250.0, RIO_Hty := 1);
   AIT503_FB : AIN_FBD := (Raw_RIO := 5384, Raw_WRIO := 6434, H_Raw_RIO := 31208, L_Raw_WRIO := 3277, H_Raw_WRIO := 16383, HEU := 1000, Hty := 1, AL := 1, SAHH := 500.0, SAH := 260.0, SAL := 250.0, RIO_Hty := 1);
   AIT504_FB : AIN_FBD := (Raw_RIO := 944, Raw_WRIO := 3355, H_Raw_RIO := 31208, L_Raw_WRIO := 3277, H_Raw_WRIO := 16383, HEU := 1200, Hty := 1, SAHH := 50.0, SAH := 40.0, RIO_Hty := 1);
   DI_DPSH_301_HIGH : BOOL;
   DI_LS_401_LOW : BOOL;
   DI_MV_501_ZSC : BOOL := 1;
   DI_MV_501_ZSO : BOOL;
   DI_MV_502_ZSC : BOOL := 1;
   DI_MV_502_ZSO : BOOL;
   DI_MV_503_ZSC : BOOL := 1;
   DI_MV_503_ZSO : BOOL;
   DI_MV_504_ZSC : BOOL := 1;
   DI_MV_504_ZSO : BOOL;
   DI_P_401_AUTO : BOOL := 1;
   DI_P_401_FAULT : BOOL;
   DI_P_401_RUN : BOOL;
   DI_P_402_AUTO : BOOL := 1;
   DI_P_402_FAULT : BOOL;
   DI_P_402_RUN : BOOL;
   DI_P_403_AUTO : BOOL := 1;
   DI_P_403_FAULT : BOOL;
   DI_P_403_RUN : BOOL;
   DI_P_404_AUTO : BOOL := 1;
   DI_P_404_FAULT : BOOL;
   DI_P_404_RUN : BOOL;
   DI_P_501_AUTO : BOOL := 1;
   DI_P_501_FAULT : BOOL;
   DI_P_501_RUN : BOOL;
   DI_P_502_AUTO : BOOL := 1;
   DI_P_502_FAULT : BOOL;
   DI_P_502_RUN : BOOL;
   DI_PSH_501_HIGH : BOOL;
   DI_PSL_501_LOW : BOOL;
   DI_RIO4_SPARE_10 : BOOL;
   DI_RIO4_SPARE_11 : BOOL;
   DI_RIO4_SPARE_12 : BOOL;
   DI_RIO4_SPARE_13 : BOOL;
   DI_RIO4_SPARE_14 : BOOL;
   DI_RIO4_SPARE_15 : BOOL;
   DI_RIO4_SPARE_16 : BOOL;
   DI_RIO4_SPARE_17 : BOOL;
   DI_RIO4_SPARE_19 : BOOL;
   DI_RIO4_SPARE_20 : BOOL;
   DI_RIO4_SPARE_21 : BOOL;
   DI_RIO4_SPARE_22 : BOOL;
   DI_RIO4_SPARE_23 : BOOL;
   DI_RIO4_SPARE_24 : BOOL;
   DI_RIO4_SPARE_25 : BOOL;
   DI_RIO4_SPARE_26 : BOOL;
   DI_RIO4_SPARE_27 : BOOL;
   DI_RIO4_SPARE_28 : BOOL;
   DI_RIO4_SPARE_29 : BOOL;
   DI_RIO4_SPARE_30 : BOOL;
   DI_RIO4_SPARE_31 : BOOL;
   DI_RIO5_SPARE_19 : BOOL;
   DI_RIO5_SPARE_20 : BOOL;
   DI_RIO5_SPARE_21 : BOOL;
   DI_RIO5_SPARE_22 : BOOL;
   DI_RIO5_SPARE_23 : BOOL;
   DI_RIO5_SPARE_24 : BOOL;
   DI_RIO5_SPARE_25 : BOOL;
   DI_RIO5_SPARE_26 : BOOL;
   DI_RIO5_SPARE_27 : BOOL;
   DI_RIO5_SPARE_28 : BOOL;
   DI_RIO5_SPARE_29 : BOOL;
   DI_RIO5_SPARE_30 : BOOL;
   DI_RIO5_SPARE_31 : BOOL;
   DI_UV_401_AUTO : BOOL := 1;
   DI_UV_401_FAULT : BOOL;
   DI_UV_401_RUN : BOOL;
   DI_UV_402_FAULT : BOOL;
   DI_UV_402_RUN : BOOL;
   DI_VSD_1_PB : BOOL;
   DI_VSD_2_PB : BOOL;
   DI_WIFI_PLC_4 : BOOL := 1;
   DI_WIFI_PLC_5 : BOOL;
   DI_WIFI_RIO_4 : BOOL;
   DI_WIFI_RIO_5 : BOOL;
   DO_MV_501_CLOSE : BOOL := 1;
   DO_MV_501_OPEN : BOOL;
   DO_MV_502_CLOSE : BOOL := 1;
   DO_MV_502_OPEN : BOOL;
   DO_MV_503_CLOSE : BOOL := 1;
   DO_MV_503_OPEN : BOOL;
   DO_MV_504_CLOSE : BOOL := 1;
   DO_MV_504_OPEN : BOOL;
   DO_P_401_START : BOOL;
   DO_P_402_START : BOOL;
   DO_P_403_START : BOOL;
   DO_P_404_START : BOOL;
   DO_RIO4_SPARE_04 : BOOL;
   DO_RIO4_SPARE_05 : BOOL;
   DO_RIO4_SPARE_06 : BOOL;
   DO_RIO4_SPARE_07 : BOOL;
   DO_RIO4_SPARE_08 : BOOL;
   DO_RIO4_SPARE_09 : BOOL;
   DO_RIO4_SPARE_10 : BOOL;
   DO_RIO4_SPARE_11 : BOOL;
   DO_RIO4_SPARE_12 : BOOL;
   DO_RIO4_SPARE_13 : BOOL;
   DO_RIO4_SPARE_14 : BOOL;
   DO_RIO4_SPARE_15 : BOOL;
   DO_RIO5_SPARE_04 : BOOL;
   DO_RIO5_SPARE_05 : BOOL;
   DO_RIO5_SPARE_06 : BOOL;
   DO_RIO5_SPARE_07 : BOOL;
   DO_RIO5_SPARE_08 : BOOL;
   DO_RIO5_SPARE_09 : BOOL;
   DO_RIO5_SPARE_10 : BOOL;
   DO_RIO5_SPARE_11 : BOOL;
   DO_RIO5_SPARE_12 : BOOL;
   DO_RIO5_SPARE_13 : BOOL;
   DO_RIO5_SPARE_14 : BOOL;
   DO_RIO5_SPARE_15 : BOOL;
   DO_UV_401_START : BOOL;
   DUMMY_AIT : AIN_UDT;
   FIT401_FB : FIT_FBD := (Raw_RIO := -19, Raw_WRIO := 3263, L_Raw_RIO := 6242, H_Raw_RIO := 31208, L_Raw_WRIO := 3277, H_Raw_WRIO := 16383, HEU := 5.0, Hty := 1, AL := 1, ALL := 1, RIO_Hty := 1);
   FIT501_FB : FIT_FBD := (Raw_RIO := 15, Raw_WRIO := 8777, H_Raw_RIO := 31208, L_Raw_WRIO := 3277, H_Raw_WRIO := 16383, HEU := 4.0, Hty := 1, AL := 1, SAHH := 3.0, SAH := 2.0, SAL := 1.0, RIO_Hty := 1);
   FIT502_FB : FIT_FBD := (Raw_RIO := -9, Raw_WRIO := 7239, L_Raw_RIO := -20, H_Raw_RIO := 31208, L_Raw_WRIO := 3277, H_Raw_WRIO := 16383, HEU := 4.0, Hty := 1, AHH := 1, AH := 1, RIO_Hty := 1);
   FIT503_FB : FIT_FBD := (Raw_RIO := -24, Raw_WRIO := 5689, L_Raw_RIO := -35, H_Raw_RIO := 31208, L_Raw_WRIO := 3277, H_Raw_WRIO := 16383, HEU := 4.0, Hty := 1, AHH := 1, AH := 1, RIO_Hty := 1, Totaliser_Enb := 1);
   FIT504_FB : FIT_FBD := (Raw_RIO := -26, Raw_WRIO := 5188, L_Raw_RIO := -15, H_Raw_RIO := 31208, L_Raw_WRIO := 3277, H_Raw_WRIO := 16383, HEU := 2.0, AL := 1, ALL := 1, SAHH := 3.5, SAH := 1.0, RIO_Hty := 1, Totaliser_Enb := 1);
   HMI_AIT401 : AIN_UDT := (Pv := -0.00070494745, AL := 1, ALL := 1, Hty := 1);
   HMI_AIT402 : AIN_UDT := (Pv := -0.0010894643, AL := 1, ALL := 1, Hty := 1);
   HMI_AIT501 : AIN_UDT := (Pv := 8.054216, AHH := 1, AH := 1, Hty := 1, Sim_PV := 8.054216);
   HMI_AIT502 : AIN_UDT := (Pv := 230.91515, SAHH := 300.0, SAH := 250.0, Hty := 1, Sim_PV := 230.91515);
   HMI_AIT503 : AIN_UDT := (Pv := 172.51987, SAHH := 500.0, SAH := 260.0, SAL := 250.0, AL := 1, Hty := 1, Sim_PV := 172.51987);
   HMI_AIT504 : AIN_UDT := (Pv := 36.298386, SAHH := 50.0, SAH := 40.0, Hty := 1, Sim_PV := 36.298386);
   HMI_FIT401 : FIT_UDT := (Pv := 0.0010243934, SAHH := 3.0, SAH := 2.0, SAL := 0.5, SALL := 0.4, Totaliser := 381.51465, AL := 1, ALL := 1, Sim_PV := 0.0010243934, Hty := 1);
   HMI_FIT501 : FIT_UDT := (Pv := 0.001922584, SAHH := 3.0, SAH := 2.0, SAL := 1.0, Totaliser := 448.75452, AL := 1, Sim_PV := 0.001922584, Hty := 1);
   HMI_FIT502 : FIT_UDT := (Pv := 0.001408992, Totaliser := 331.85107, AHH := 1, AH := 1, Sim_PV := 0.001408992, Hty := 1);
   HMI_FIT503 : FIT_UDT := (Pv := 0.0014083155, Totaliser := 52.980667, AHH := 1, AH := 1, Sim_PV := 0.0014083155, Hty := 1);
   HMI_FIT504 : FIT_UDT := (SAHH := 3.5, SAH := 1.0, Totaliser := 129.2501, AL := 1, ALL := 1);
   HMI_FLUSHING_MIN : INT;
   HMI_FLUSHING_MIN_SP : INT := 1;
   HMI_HIGH_RO_MAX_SPEED : REAL;
   HMI_HIGH_RO_MIN_SPEED : REAL := 10.0;
   HMI_HPP_Q_MAX_M3H : REAL := 2.0;
   HMI_HPP_Q_SET_M3H : REAL := 1.25;
   HMI_LIT401 : AIN_UDT := (Pv := -0.0005767752, AL := 1, ALL := 1, Hty := 1);
   HMI_LS401 : SWITCH_UDT;
   HMI_MIN_RO_VSD_SPEED : REAL := 3.125;
   HMI_MV501 : MV_UDT := (Cmd := 1, Status := 1, Reset := 1, Auto := 1, Avl := 1);
   HMI_MV501_TIMEOUT_TM : INT;
   HMI_MV502 : MV_UDT := (Cmd := 1, Status := 1, Reset := 1, Auto := 1, Avl := 1);
   HMI_MV502_TIMEOUT_TM : INT;
   HMI_MV503 : MV_UDT := (Cmd := 1, Status := 1, Reset := 1, Auto := 1, Avl := 1);
   HMI_MV503_TIMEOUT_TM : INT;
   HMI_MV504 : MV_UDT := (Cmd := 1, Status := 1, Reset := 1, Auto := 1, Avl := 1);
   HMI_MV504_TIMEOUT_TM : INT;
   HMI_NAHSO3_ORP_DOSING : DOSING_SETPOINT_UDT;
   HMI_P401 : PMP_UDT := (Status := 2, Remote := 1, Permissive := -1);
   HMI_P402 : PMP_UDT := (Status := 1, Remote := 1, Permissive := -1);
   HMI_P403 : PMP_UDT := (Status := 1, Remote := 1, Permissive := -1);
   HMI_P404 : PMP_UDT := (Status := 1, Remote := 1, Permissive := -1);
   HMI_P4_PERMISSIVE : BOOL;
   HMI_P4_STATE : INT;
   HMI_P501 : VSD_UDT := (Cmd := 1, Status := 1, Total_RunMin := 17445.0, Total_RunHr := 290.75, Remote := 1, Auto := 1, Avl := 1, Speed_Command := 10.0, Permissive := -2, SD := 1, Reset := 1, Reset_RunHr := 1);
   HMI_P501_MSG : PRECONDITION_UDT := (PERMISSIVE2 := 1, PERMISSIVE3 := 1);
   HMI_P502 : VSD_UDT := (Cmd := 1, Status := 1, RunMin := 409.0, Total_RunMin := 409.0, RunHr := 6.8166666, Total_RunHr := 6.8166666, Remote := 1, Auto := 1, Avl := 1, Drive_Ready := 1, Speed_Command := 35.0, Permissive := -8, SD := 5, Reset := 1);
   HMI_P502_MSG : PRECONDITION_UDT;
   HMI_P5_PERMISSIVE : AUTOINP_UDT := (ON := 1);
   HMI_P5_SD_FLUSHING_DONE : AUTOINP_UDT;
   HMI_P5_STATE : INT := 1;
   HMI_P_NAHSO3_ORP_DUTY : Duty2_UDT;
   HMI_P_RO_FEED_DUTY : Duty2_UDT := (Selection := 1);
   HMI_P_RO_HIGH_DUTY : Duty2_UDT := (Selection := 1);
   HMI_P_UF_FEED_DUTY : Duty2_UDT;
   HMI_PERMEATE_COND_SP : REAL := 300.0;
   HMI_PERMEATE_FLOW_SP : REAL;
   HMI_PIT501 : AIN_UDT := (Pv := 11.551525, SAHH := 350.0, SAH := 280.0, Hty := 1, Sim_PV := 11.551525);
   HMI_PIT501_SP_1 : REAL;
   HMI_PIT501_SP_2 : REAL;
   HMI_PIT502 : AIN_UDT := (AHH := 1, AH := 1, AL := 1, ALL := 1);
   HMI_PIT503 : AIN_UDT := (Pv := 6.440656, AHH := 1, AH := 1, Hty := 1, Sim_PV := 6.440656);
   HMI_PLANT : PLANT_UDT;
   HMI_PLANT_AUTO : PLANT_AUTO_UDT;
   HMI_PLANT_PERMISSIVE : BOOL := 1;
   HMI_PLANT_RESET : PLANT_AUTO_UDT;
   HMI_PSH501 : SWITCH_UDT;
   HMI_PSL501 : SWITCH_UDT;
   HMI_RAMPING_RATE_PER_SEC : REAL := 1.5;
   HMI_RO_HIGH_PUMP_SHUTDOWN : BOOL;
   HMI_RO_HPP_SD : AUTOINP_UDT;
   HMI_RO_SD_FLUSHING_MIN : INT;
   HMI_RO_SD_FLUSHING_MIN_SP : INT := 1;
   HMI_RO_TMP : REAL := 9.028133;
   HMI_SHUTDOWN_FLUSHING : AUTOINP_UDT;
   HMI_START_PLANT : BOOL;
   HMI_UV401 : UV_UDT := (Cmd := 1, Status := 1, RunMin := 15329.0, Total_RunMin := 15329.0, RunHr := 255.48334, Total_RunHr := 255.48334, Remote := 1, Auto := 1, Avl := 1, Permissive := -4, Reset := 1);
   HMI_VSD_HIGH_SPEED : REAL := 30.0;
   HMI_VSD_MIN_SPEED : REAL := 10.0;
   HMI_VSD_RATE : REAL;
   HMI_WIFI : WIFI_UDT;
   LIT401_FB : AIN_FBD := (Raw_RIO := -9, Raw_WRIO := 3269, H_Raw_RIO := 31208, L_Raw_WRIO := 3277, H_Raw_WRIO := 16383, HEU := 2, Hty := 1, AL := 1, ALL := 1, RIO_Hty := 1);
   LIT401_FB_01 : AIN_FBD;
   Logix_Status : Logix_Status_FP := (Sts_MinorFaultEvents := 1, Sts_MinorFaultBits := 16, Set_FaceplateAnimation := 90, Val_ProductCode := 92, MemoryTemp[0] := 5, MemoryTemp[1] := 1, MemoryTemp[3] := 27596, MemoryTemp[4] := 3, MemoryTemp[5] := -23178, MemoryTemp[6] := 6, MemoryTemp[9] := 2, MemoryTemp[11] := -4608, MemoryTemp[12] := 3, MemoryTemp[14] := 8, MemoryTemp[17] := 5, MemoryTemp[21] := 6, MemoryTemp[23] := 26636, MemoryTemp[24] := 3, MemoryTemp[25] := 7, MemoryTemp[27] := 19904, MemoryTemp[28] := 6, Val_raw_data := 12640, Sts_IO_LED_raw := 2, Sts_ProductCode := 92, MemoryRequestData[0] := 5, MemoryRequestData[2] := 1, MemoryRequestData[4] := 2, MemoryRequestData[6] := 5, MemoryRequestData[8] := 6, MemoryRequestData[10] := 7, Sts_Run := 1, Sts_KS_in_remote := 1, Sts_Ladder_Working := 1, Set_Controller_Description := 'P5: Rerverse Osmosis System', UpdateDelayTimer.PRE := 1000, UpdateDelayTimer.ACC := 470, UpdateDelayTimer.EN := 1, UpdateDelayTimer.TT := 1, Val_MFS.timelow := 71751885, Val_MFS.timehigh := 206334, Val_MFS.type := 3, Val_MFS.code := 20, Val_MFS.info[1] := 1, Sts_IO_LED.FlashingGreen := 1, Sts_Battery_LED.Off := 1, MemoryData.Free_Mem_IO := 896816, MemoryData.Free_Mem_DT := 1742296, MemoryData.Total_Mem_IO := 1030144, MemoryData.Total_Mem_DT := 2097152, MemoryData.Biggest_IO_Mem_Size_Ava := 892976, MemoryData.Biggest_DT_Mem_Size_Ava := 1652480);
   LS401_FB : SWITCH_FBD;
   Memory_Message : MESSAGE;
        MessageParameters(ServiceCode := 16#0003, LocalElement := Logix_Status.MemoryRequestData[0], DestinationTag := Logix_Status.MemoryTemp[0], ...)
   MV501_FB : MV_FBD := (Auto := 1, Cmd_Close := 1, Open_TM := 15, ZSC := 1, Close_TM := 15);
   MV502_FB : MV_FBD := (Auto := 1, Cmd_Close := 1, Open_TM := 15, ZSC := 1, Close_TM := 15);
   MV503_FB : MV_FBD := (Auto := 1, Cmd_Close := 1, Open_TM := 15, ZSC := 1, Close_TM := 15);
   MV504_FB : MV_FBD := (Auto := 1, Cmd_Close := 1, Open_TM := 15, ZSC := 1, Close_TM := 15);
   P401_FB : PMP_FBD := (Remote := 1, Start_TM := 3, Stop_TM := 3, Permissive := -1);
   P402_FB : PMP_FBD := (Remote := 1, Start_TM := 3, Stop_TM := 3, Permissive := -1);
   P403_FB : PMP_FBD := (Remote := 1, Start_TM := 3, Stop_TM := 3, Permissive := -1);
   P404_FB : PMP_FBD := (Remote := 1, Start_TM := 3, Stop_TM := 3, Permissive := -1);
   P4_FIT401_MSG : MESSAGE;
        MessageParameters(ServiceCode := 16#004c, LocalElement := HMI_FIT401, ...)
   P4_P4012_MSG : MESSAGE;
        MessageParameters(ServiceCode := 16#004c, LocalElement := HMI_P_RO_FEED_DUTY, ...)
   P4_RO_FEED_SD_MSG : MESSAGE;
        MessageParameters(ServiceCode := 16#004d, LocalElement := HMI_RO_HPP_SD, ...)
   P4_UV401_MSG : MESSAGE;
        MessageParameters(ServiceCode := 16#004c, LocalElement := HMI_UV401, ...)
   P501_FB : VSD_FBD := (Avl := 1, Total_RunHr := 290.75, Auto := 1, Remote := 1, Start_TM := 20, Stop_TM := 20, Rst := 1, Rst_RunHr := 1, AutoSpeed := 10.0, Speed_Cmd := 10.0, Permissive := -2, Shutdown := 1);
   P502_FB : VSD_FBD := (Avl := 1, RunHr := 6.8166666, Total_RunHr := 6.8166666, Rdy := 1, Auto := 1, Remote := 1, Start_TM := 20, Stop_TM := 20, Rst := 1, AutoSpeed := 10.0, Speed_Cmd := 35.0, Permissive := -8, Shutdown := 5);
   P_NAHSO3_ORP_DUTY_FB : Duty2_FBD;
   P_RO_FEED_DUTY_FB : Duty2_FBD;
   P_RO_HIGH_DUTY_FB : Duty2_FBD := (Selection := 1);
   PIT501_FB : AIN_FBD := (Raw_RIO := 718, Raw_WRIO := 10198, H_Raw_RIO := 31208, L_Raw_WRIO := 3277, H_Raw_WRIO := 16383, HEU := 500, Hty := 1, SAHH := 350.0, SAH := 280.0, RIO_Hty := 1);
   PIT502_FB : AIN_FBD := (Raw_RIO := -21, Raw_WRIO := 3289, L_Raw_RIO := -5, H_Raw_RIO := 31208, L_Raw_WRIO := 3277, H_Raw_WRIO := 16383, HEU := 500, AHH := 1, AH := 1, AL := 1, ALL := 1, RIO_Hty := 1);
   PIT503_FB : AIN_FBD := (Raw_RIO := 402, Raw_WRIO := 8615, H_Raw_RIO := 31208, L_Raw_WRIO := 3277, H_Raw_WRIO := 16383, HEU := 500, Hty := 1, AHH := 1, AH := 1, RIO_Hty := 1);
   PSH501_FB : SWITCH_FBD;
   PSL501_FB : SWITCH_FBD;
   R_TRIG : FBD_ONESHOT;
   R_TRIG_MIN : FBD_ONESHOT;
   REDUNDANT_STATUS : RED_STAT := (Redundancy_status_of_the_controller := 2, Redundancy_state_of_the_partner := 8);
   RTRIG_SEC : FBD_ONESHOT;
   RTRIG_SEC1 : FBD_ONESHOT;
   TEST : BOOL;
   TEST_MIN : DINT := 457528;
   TEST_SEC : DINT;
   TEST_SEC1 : DINT;
   TON : FBD_TIMER := (TimerEnable := 1, PRE := 1000, ACC := 963, EN := 1, TT := 1);
   TON_FIT401_TM : FBD_TIMER := (PRE := 3000);
   TON_MIN : FBD_TIMER := (TimerEnable := 1, PRE := 60000, ACC := 26318, EN := 1, TT := 1);
   TON_SEC : FBD_TIMER := (TimerEnable := 1, PRE := 1000, ACC := 66, EN := 1, TT := 1);
   TON_SEC1 : FBD_TIMER := (TimerEnable := 1, PRE := 1000, ACC := 117, EN := 1, TT := 1);
   UV401_FB : UV_FBD := (AutoInp := 1, Remote := 1, Start_TM := 3, Stop_TM := 3, Permissive := -1);
   W_AI_AIT_401_HRDNSS : INT := 3266;
   W_AI_AIT_401_HRDNSS_HTY : BOOL;
   W_AI_AIT_402_ORP : INT := 3268;
   W_AI_AIT_402_ORP_HTY : BOOL;
   W_AI_AIT_501_PH : INT := 10247;
   W_AI_AIT_501_PH_HTY : BOOL;
   W_AI_AIT_502_ORP : INT := 6637;
   W_AI_AIT_502_ORP_HTY : BOOL;
   W_AI_AIT_503_COND : INT := 6434;
   W_AI_AIT_503_COND_HTY : BOOL;
   W_AI_AIT_504_COND : INT := 3355;
   W_AI_AIT_504_COND_HTY : BOOL;
   W_AI_FIT_401_FLOW : INT := 3263;
   W_AI_FIT_401_FLOW_HTY : BOOL;
   W_AI_FIT_501_FLOW : INT := 8777;
   W_AI_FIT_501_FLOW_HTY : BOOL;
   W_AI_FIT_502_FLOW : INT := 7239;
   W_AI_FIT_502_FLOW_HTY : BOOL;
   W_AI_FIT_503_FLOW : INT := 5689;
   W_AI_FIT_503_FLOW_HTY : BOOL;
   W_AI_FIT_504_FLOW : INT := 5188;
   W_AI_FIT_504_FLOW_HTY : BOOL;
   W_AI_LIT_301_LEVEL : INT;
   W_AI_LIT_301_LEVEL_HTY : BOOL;
   W_AI_LIT_401_LEVEL : INT := 3269;
   W_AI_LIT_401_LEVEL_HTY : BOOL;
   W_AI_PIT_501_PRESS : INT := 10198;
   W_AI_PIT_501_PRESS_HTY : BOOL;
   W_AI_PIT_502_PRESS : INT := 3289;
   W_AI_PIT_502_PRESS_HTY : BOOL;
   W_AI_PIT_503_PRESS : INT := 8615;
   W_AI_PIT_503_PRESS_HTY : BOOL;
   W_AI_RIO4_SPARE_03_HTY : BOOL;
   W_AI_W_AIT_501_PH : INT;
   W_AI_W_AIT_501_PH_HTY : BOOL;
   W_AI_W_AIT_502_ORP : INT;
   W_AI_W_AIT_502_ORP_HTY : BOOL;
   W_AI_W_AIT_503_COND : INT;
   W_AI_W_AIT_503_COND_HTY : BOOL;
   W_AI_W_AIT_504_COND : INT;
   W_AI_W_AIT_504_COND_HTY : BOOL;
   XXX : DINT;
END_VAR

PROGRAM MainProgram   (* main routine MainRoutine *)
VAR
   DO_LED_RED : BOOL;
   Duty2_FBD_01 : Duty2_FBD;
   FIT401_LL_STATE : DINT := 1;
   FIT401_LL_STATE4 : DINT;
   MV_FBD_01 : MV_FBD;
   P401_OFF_STATE : DINT;
   P401_ON_STATE : DINT := 2;
   SEC_COUNT : DINT;
   SEC_COUNT1 : DINT := 1;
   SWITCH_FBD_01 : SWITCH_FBD;
   UV401_OFF_STATE : DINT := 2;
   VSD_FBD_01 : VSD_FBD;
END_VAR

ROUTINE High_Pressure_RO   (* function block diagram *)
   SHEET 1
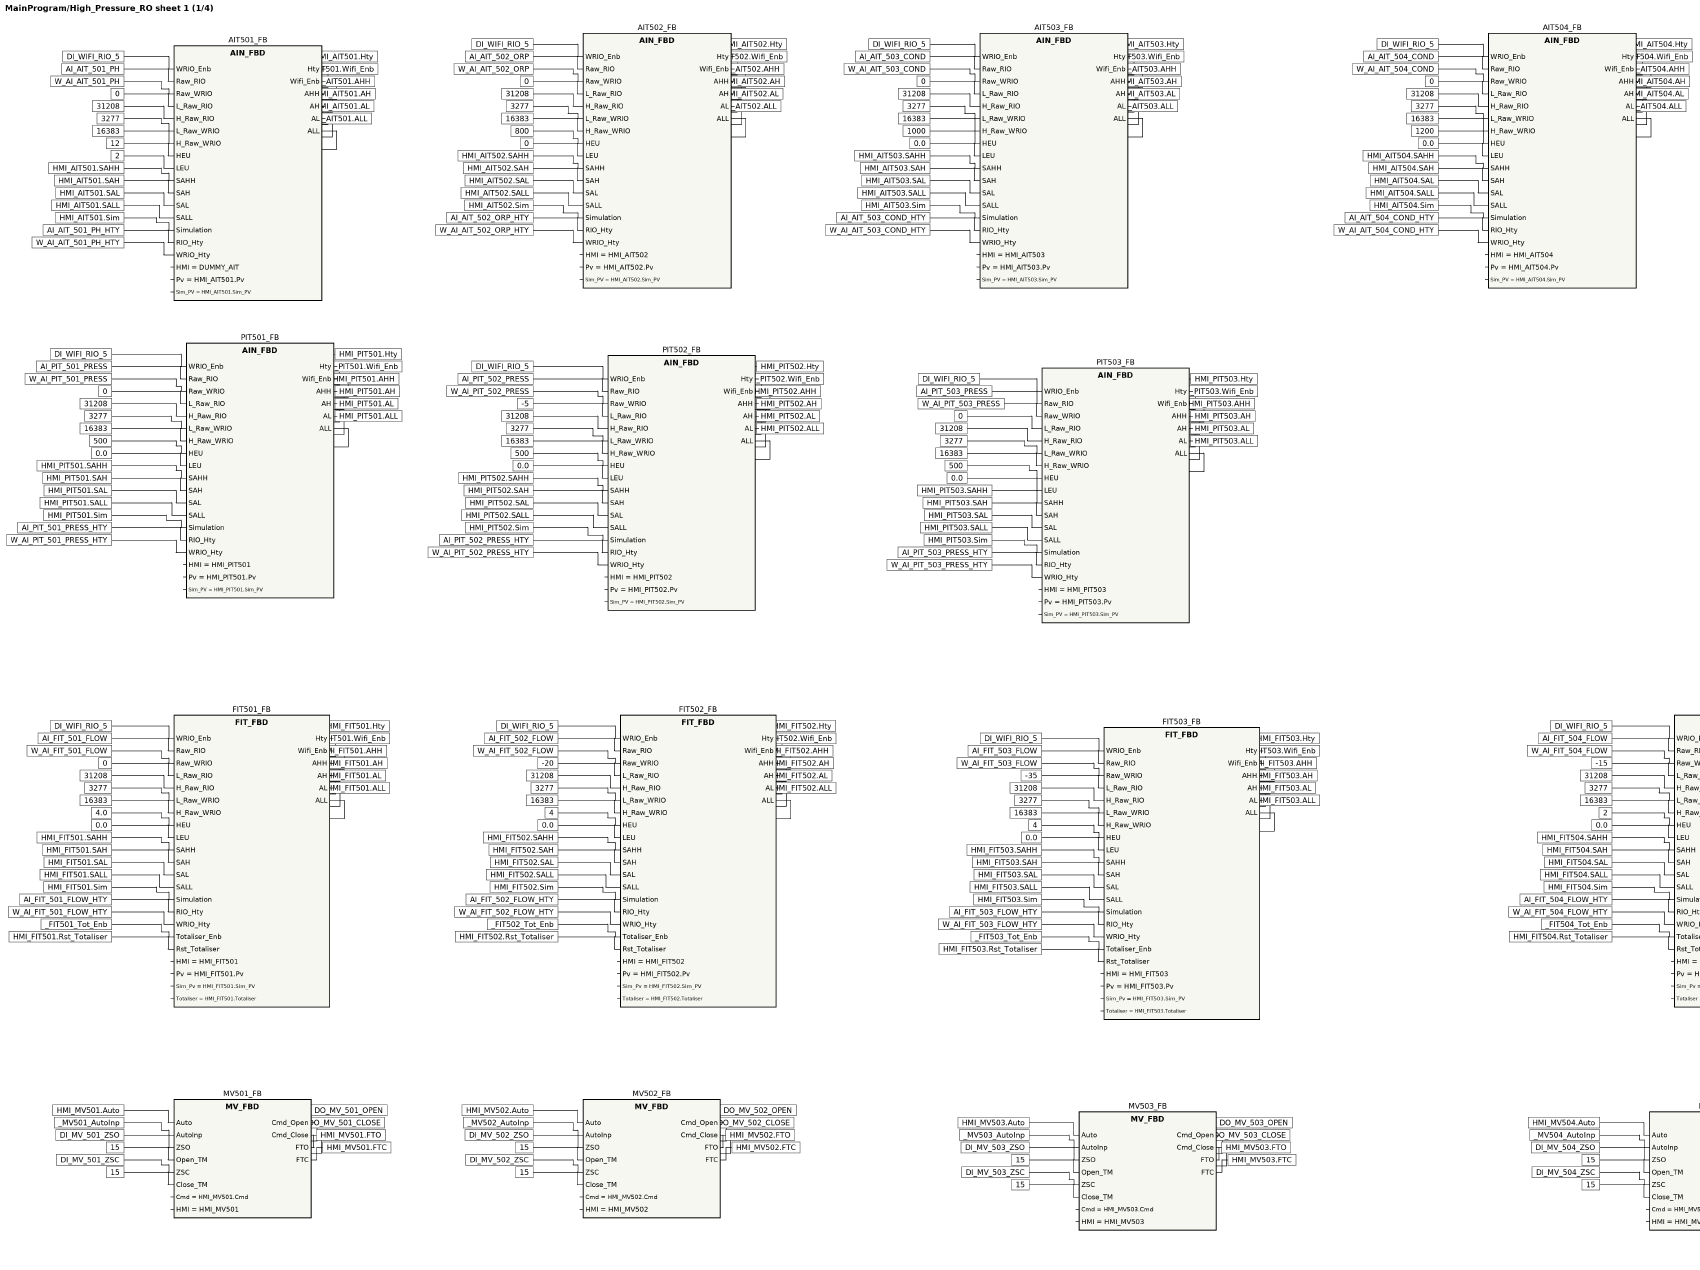
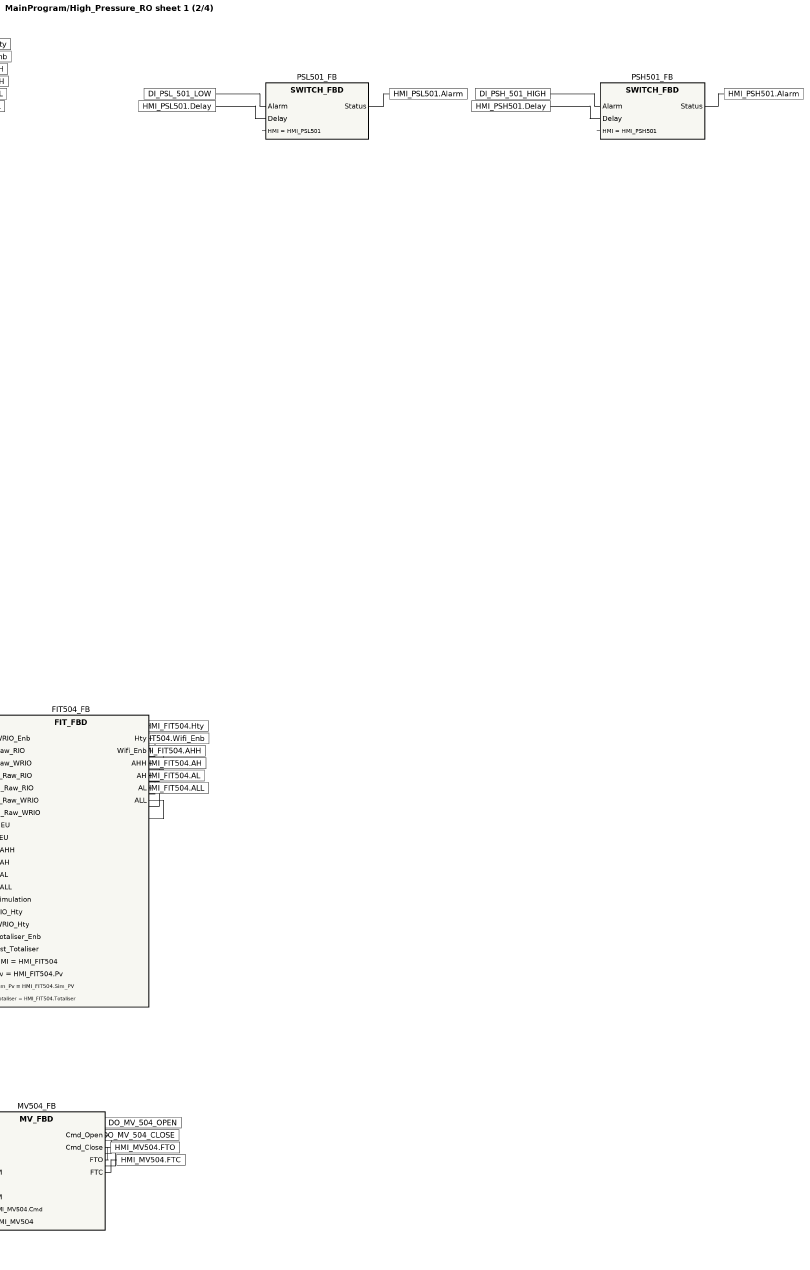
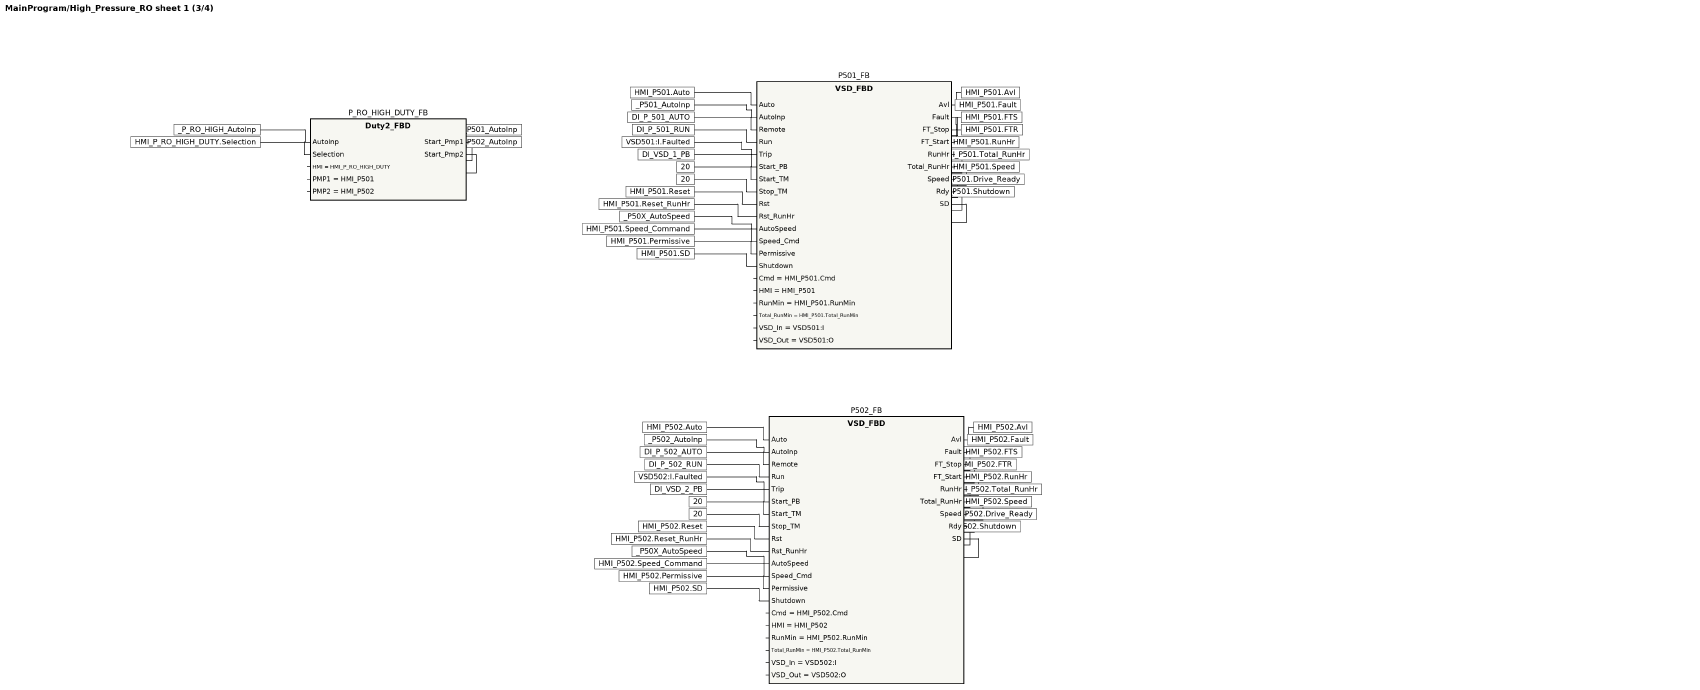
   AIT501_FB : AIN_FBD(WRIO_Enb := DI_WIFI_RIO_5, Raw_RIO := AI_AIT_501_PH, Raw_WRIO := W_AI_AIT_501_PH, L_Raw_RIO := 0, H_Raw_RIO := 31208, L_Raw_WRIO := 3277, H_Raw_WRIO := 16383, HEU := 12, LEU := 2, SAHH := HMI_AIT501.SAHH, SAH := HMI_AIT501.SAH, SAL := HMI_AIT501.SAL, SALL := HMI_AIT501.SALL, Simulation := HMI_AIT501.Sim, RIO_Hty := AI_AIT_501_PH_HTY, WRIO_Hty := W_AI_AIT_501_PH_HTY, HMI := DUMMY_AIT, Pv := HMI_AIT501.Pv, Sim_PV := HMI_AIT501.Sim_PV);
   FIT501_FB : FIT_FBD(WRIO_Enb := DI_WIFI_RIO_5, Raw_RIO := AI_FIT_501_FLOW, Raw_WRIO := W_AI_FIT_501_FLOW, L_Raw_RIO := 0, H_Raw_RIO := 31208, L_Raw_WRIO := 3277, H_Raw_WRIO := 16383, HEU := 4.0, LEU := 0.0, SAHH := HMI_FIT501.SAHH, SAH := HMI_FIT501.SAH, SAL := HMI_FIT501.SAL, SALL := HMI_FIT501.SALL, Simulation := HMI_FIT501.Sim, RIO_Hty := AI_FIT_501_FLOW_HTY, WRIO_Hty := W_AI_FIT_501_FLOW_HTY, Totaliser_Enb := _FIT501_Tot_Enb, Rst_Totaliser := HMI_FIT501.Rst_Totaliser, HMI := HMI_FIT501, Pv := HMI_FIT501.Pv, Sim_Pv := HMI_FIT501.Sim_PV, Totaliser := HMI_FIT501.Totaliser);
   MV501_FB : MV_FBD(Auto := HMI_MV501.Auto, AutoInp := _MV501_AutoInp, ZSO := DI_MV_501_ZSO, Open_TM := 15, ZSC := DI_MV_501_ZSC, Close_TM := 15, Cmd := HMI_MV501.Cmd, HMI := HMI_MV501);
   PIT501_FB : AIN_FBD(WRIO_Enb := DI_WIFI_RIO_5, Raw_RIO := AI_PIT_501_PRESS, Raw_WRIO := W_AI_PIT_501_PRESS, L_Raw_RIO := 0, H_Raw_RIO := 31208, L_Raw_WRIO := 3277, H_Raw_WRIO := 16383, HEU := 500, LEU := 0.0, SAHH := HMI_PIT501.SAHH, SAH := HMI_PIT501.SAH, SAL := HMI_PIT501.SAL, SALL := HMI_PIT501.SALL, Simulation := HMI_PIT501.Sim, RIO_Hty := AI_PIT_501_PRESS_HTY, WRIO_Hty := W_AI_PIT_501_PRESS_HTY, HMI := HMI_PIT501, Pv := HMI_PIT501.Pv, Sim_PV := HMI_PIT501.Sim_PV);
   HMI_AIT501.Wifi_Enb := AIT501_FB.Wifi_Enb;
   HMI_AIT501.AHH := AIT501_FB.AHH;
   HMI_AIT501.ALL := AIT501_FB.ALL;
   HMI_FIT501.Wifi_Enb := FIT501_FB.Wifi_Enb;
   DO_MV_501_CLOSE := MV501_FB.Cmd_Close;
   HMI_AIT501.Hty := AIT501_FB.Hty;
   HMI_AIT501.AH := AIT501_FB.AH;
   HMI_AIT501.AL := AIT501_FB.AL;
   DO_MV_501_OPEN := MV501_FB.Cmd_Open;
   P_RO_HIGH_DUTY_FB : Duty2_FBD(AutoInp := _P_RO_HIGH_AutoInp, Selection := HMI_P_RO_HIGH_DUTY.Selection, HMI := HMI_P_RO_HIGH_DUTY, PMP1 := HMI_P501, PMP2 := HMI_P502);
   HMI_PIT501.Wifi_Enb := PIT501_FB.Wifi_Enb;
   HMI_FIT501.AHH := FIT501_FB.AHH;
   HMI_MV501.FTO := MV501_FB.FTO;
   HMI_FIT501.Hty := FIT501_FB.Hty;
   HMI_FIT501.AH := FIT501_FB.AH;
   HMI_FIT501.AL := FIT501_FB.AL;
   HMI_FIT501.ALL := FIT501_FB.ALL;
   HMI_MV501.FTC := MV501_FB.FTC;
   HMI_PIT501.AHH := PIT501_FB.AHH;
   HMI_PIT501.Hty := PIT501_FB.Hty;
   HMI_PIT501.AH := PIT501_FB.AH;
   HMI_PIT501.AL := PIT501_FB.AL;
   HMI_PIT501.ALL := PIT501_FB.ALL;
   _P501_AutoInp := P_RO_HIGH_DUTY_FB.Start_Pmp1;
   _P502_AutoInp := P_RO_HIGH_DUTY_FB.Start_Pmp2;
   AIT502_FB : AIN_FBD(WRIO_Enb := DI_WIFI_RIO_5, Raw_RIO := AI_AIT_502_ORP, Raw_WRIO := W_AI_AIT_502_ORP, L_Raw_RIO := 0, H_Raw_RIO := 31208, L_Raw_WRIO := 3277, H_Raw_WRIO := 16383, HEU := 800, LEU := 0, SAHH := HMI_AIT502.SAHH, SAH := HMI_AIT502.SAH, SAL := HMI_AIT502.SAL, SALL := HMI_AIT502.SALL, Simulation := HMI_AIT502.Sim, RIO_Hty := AI_AIT_502_ORP_HTY, WRIO_Hty := W_AI_AIT_502_ORP_HTY, HMI := HMI_AIT502, Pv := HMI_AIT502.Pv, Sim_PV := HMI_AIT502.Sim_PV);
   MV502_FB : MV_FBD(Auto := HMI_MV502.Auto, AutoInp := _MV502_AutoInp, ZSO := DI_MV_502_ZSO, Open_TM := 15, ZSC := DI_MV_502_ZSC, Close_TM := 15, Cmd := HMI_MV502.Cmd, HMI := HMI_MV502);
   PIT502_FB : AIN_FBD(WRIO_Enb := DI_WIFI_RIO_5, Raw_RIO := AI_PIT_502_PRESS, Raw_WRIO := W_AI_PIT_502_PRESS, L_Raw_RIO := -5, H_Raw_RIO := 31208, L_Raw_WRIO := 3277, H_Raw_WRIO := 16383, HEU := 500, LEU := 0.0, SAHH := HMI_PIT502.SAHH, SAH := HMI_PIT502.SAH, SAL := HMI_PIT502.SAL, SALL := HMI_PIT502.SALL, Simulation := HMI_PIT502.Sim, RIO_Hty := AI_PIT_502_PRESS_HTY, WRIO_Hty := W_AI_PIT_502_PRESS_HTY, HMI := HMI_PIT502, Pv := HMI_PIT502.Pv, Sim_PV := HMI_PIT502.Sim_PV);
   FIT502_FB : FIT_FBD(WRIO_Enb := DI_WIFI_RIO_5, Raw_RIO := AI_FIT_502_FLOW, Raw_WRIO := W_AI_FIT_502_FLOW, L_Raw_RIO := -20, H_Raw_RIO := 31208, L_Raw_WRIO := 3277, H_Raw_WRIO := 16383, HEU := 4, LEU := 0.0, SAHH := HMI_FIT502.SAHH, SAH := HMI_FIT502.SAH, SAL := HMI_FIT502.SAL, SALL := HMI_FIT502.SALL, Simulation := HMI_FIT502.Sim, RIO_Hty := AI_FIT_502_FLOW_HTY, WRIO_Hty := W_AI_FIT_502_FLOW_HTY, Totaliser_Enb := _FIT502_Tot_Enb, Rst_Totaliser := HMI_FIT502.Rst_Totaliser, HMI := HMI_FIT502, Pv := HMI_FIT502.Pv, Sim_Pv := HMI_FIT502.Sim_PV, Totaliser := HMI_FIT502.Totaliser);
   HMI_AIT502.Wifi_Enb := AIT502_FB.Wifi_Enb;
   HMI_AIT502.AHH := AIT502_FB.AHH;
   HMI_AIT502.ALL := AIT502_FB.ALL;
   DO_MV_502_CLOSE := MV502_FB.Cmd_Close;
   HMI_AIT502.Hty := AIT502_FB.Hty;
   HMI_AIT502.AH := AIT502_FB.AH;
   HMI_AIT502.AL := AIT502_FB.AL;
   DO_MV_502_OPEN := MV502_FB.Cmd_Open;
   HMI_MV502.FTO := MV502_FB.FTO;
   HMI_MV502.FTC := MV502_FB.FTC;
   HMI_PIT502.Wifi_Enb := PIT502_FB.Wifi_Enb;
   HMI_PIT502.AHH := PIT502_FB.AHH;
   HMI_FIT502.Wifi_Enb := FIT502_FB.Wifi_Enb;
   HMI_PIT502.Hty := PIT502_FB.Hty;
   HMI_PIT502.AH := PIT502_FB.AH;
   HMI_PIT502.AL := PIT502_FB.AL;
   HMI_PIT502.ALL := PIT502_FB.ALL;
   P501_FB : VSD_FBD(Auto := HMI_P501.Auto, AutoInp := _P501_AutoInp, Remote := DI_P_501_AUTO, Run := DI_P_501_RUN, Trip := VSD501:I.Faulted, Start_PB := DI_VSD_1_PB, Start_TM := 20, Stop_TM := 20, Rst := HMI_P501.Reset, Rst_RunHr := HMI_P501.Reset_RunHr, AutoSpeed := _P50X_AutoSpeed, Speed_Cmd := HMI_P501.Speed_Command, Permissive := HMI_P501.Permissive, Shutdown := HMI_P501.SD, Cmd := HMI_P501.Cmd, HMI := HMI_P501, RunMin := HMI_P501.RunMin, Total_RunMin := HMI_P501.Total_RunMin, VSD_In := VSD501:I, VSD_Out := VSD501:O);
   HMI_FIT502.AHH := FIT502_FB.AHH;
   HMI_FIT502.Hty := FIT502_FB.Hty;
   HMI_FIT502.AH := FIT502_FB.AH;
   HMI_FIT502.AL := FIT502_FB.AL;
   HMI_FIT502.ALL := FIT502_FB.ALL;
   P502_FB : VSD_FBD(Auto := HMI_P502.Auto, AutoInp := _P502_AutoInp, Remote := DI_P_502_AUTO, Run := DI_P_502_RUN, Trip := VSD502:I.Faulted, Start_PB := DI_VSD_2_PB, Start_TM := 20, Stop_TM := 20, Rst := HMI_P502.Reset, Rst_RunHr := HMI_P502.Reset_RunHr, AutoSpeed := _P50X_AutoSpeed, Speed_Cmd := HMI_P502.Speed_Command, Permissive := HMI_P502.Permissive, Shutdown := HMI_P502.SD, Cmd := HMI_P502.Cmd, HMI := HMI_P502, RunMin := HMI_P502.RunMin, Total_RunMin := HMI_P502.Total_RunMin, VSD_In := VSD502:I, VSD_Out := VSD502:O);
   HMI_P501.Drive_Ready := P501_FB.Rdy;
   HMI_P501.Shutdown := P501_FB.SD;
   HMI_P501.Total_RunHr := P501_FB.Total_RunHr;
   HMI_P502.Shutdown := P502_FB.SD;
   HMI_P502.Drive_Ready := P502_FB.Rdy;
   HMI_P501.RunHr := P501_FB.RunHr;
   HMI_P501.Speed := P501_FB.Speed;
   HMI_P502.Total_RunHr := P502_FB.Total_RunHr;
   HMI_P501.Fault := P501_FB.Fault;
   HMI_P502.FTR := P502_FB.FT_Start;
   HMI_P501.Avl := P501_FB.Avl;
   HMI_P501.FTS := P501_FB.FT_Stop;
   HMI_P501.FTR := P501_FB.FT_Start;
   HMI_P502.FTS := P502_FB.FT_Stop;
   HMI_P502.RunHr := P502_FB.RunHr;
   HMI_P502.Speed := P502_FB.Speed;
   HMI_P502.Fault := P502_FB.Fault;
   HMI_P502.Avl := P502_FB.Avl;
   AIT503_FB : AIN_FBD(WRIO_Enb := DI_WIFI_RIO_5, Raw_RIO := AI_AIT_503_COND, Raw_WRIO := W_AI_AIT_503_COND, L_Raw_RIO := 0, H_Raw_RIO := 31208, L_Raw_WRIO := 3277, H_Raw_WRIO := 16383, HEU := 1000, LEU := 0.0, SAHH := HMI_AIT503.SAHH, SAH := HMI_AIT503.SAH, SAL := HMI_AIT503.SAL, SALL := HMI_AIT503.SALL, Simulation := HMI_AIT503.Sim, RIO_Hty := AI_AIT_503_COND_HTY, WRIO_Hty := W_AI_AIT_503_COND_HTY, HMI := HMI_AIT503, Pv := HMI_AIT503.Pv, Sim_PV := HMI_AIT503.Sim_PV);
   PIT503_FB : AIN_FBD(WRIO_Enb := DI_WIFI_RIO_5, Raw_RIO := AI_PIT_503_PRESS, Raw_WRIO := W_AI_PIT_503_PRESS, L_Raw_RIO := 0, H_Raw_RIO := 31208, L_Raw_WRIO := 3277, H_Raw_WRIO := 16383, HEU := 500, LEU := 0.0, SAHH := HMI_PIT503.SAHH, SAH := HMI_PIT503.SAH, SAL := HMI_PIT503.SAL, SALL := HMI_PIT503.SALL, Simulation := HMI_PIT503.Sim, RIO_Hty := AI_PIT_503_PRESS_HTY, WRIO_Hty := W_AI_PIT_503_PRESS_HTY, HMI := HMI_PIT503, Pv := HMI_PIT503.Pv, Sim_PV := HMI_PIT503.Sim_PV);
   MV503_FB : MV_FBD(Auto := HMI_MV503.Auto, AutoInp := _MV503_AutoInp, ZSO := DI_MV_503_ZSO, Open_TM := 15, ZSC := DI_MV_503_ZSC, Close_TM := 15, Cmd := HMI_MV503.Cmd, HMI := HMI_MV503);
   HMI_AIT503.Wifi_Enb := AIT503_FB.Wifi_Enb;
   FIT503_FB : FIT_FBD(WRIO_Enb := DI_WIFI_RIO_5, Raw_RIO := AI_FIT_503_FLOW, Raw_WRIO := W_AI_FIT_503_FLOW, L_Raw_RIO := -35, H_Raw_RIO := 31208, L_Raw_WRIO := 3277, H_Raw_WRIO := 16383, HEU := 4, LEU := 0.0, SAHH := HMI_FIT503.SAHH, SAH := HMI_FIT503.SAH, SAL := HMI_FIT503.SAL, SALL := HMI_FIT503.SALL, Simulation := HMI_FIT503.Sim, RIO_Hty := AI_FIT_503_FLOW_HTY, WRIO_Hty := W_AI_FIT_503_FLOW_HTY, Totaliser_Enb := _FIT503_Tot_Enb, Rst_Totaliser := HMI_FIT503.Rst_Totaliser, HMI := HMI_FIT503, Pv := HMI_FIT503.Pv, Sim_Pv := HMI_FIT503.Sim_PV, Totaliser := HMI_FIT503.Totaliser);
   HMI_AIT503.AHH := AIT503_FB.AHH;
   HMI_AIT503.ALL := AIT503_FB.ALL;
   HMI_AIT503.Hty := AIT503_FB.Hty;
   HMI_AIT503.AH := AIT503_FB.AH;
   HMI_AIT503.AL := AIT503_FB.AL;
   HMI_PIT503.Wifi_Enb := PIT503_FB.Wifi_Enb;
   HMI_PIT503.AHH := PIT503_FB.AHH;
   HMI_PIT503.Hty := PIT503_FB.Hty;
   HMI_PIT503.AH := PIT503_FB.AH;
   HMI_PIT503.AL := PIT503_FB.AL;
   HMI_PIT503.ALL := PIT503_FB.ALL;
   DO_MV_503_CLOSE := MV503_FB.Cmd_Close;
   DO_MV_503_OPEN := MV503_FB.Cmd_Open;
   HMI_MV503.FTO := MV503_FB.FTO;
   HMI_MV503.FTC := MV503_FB.FTC;
   HMI_FIT503.Wifi_Enb := FIT503_FB.Wifi_Enb;
   HMI_FIT503.AHH := FIT503_FB.AHH;
   HMI_FIT503.Hty := FIT503_FB.Hty;
   HMI_FIT503.AH := FIT503_FB.AH;
   HMI_FIT503.AL := FIT503_FB.AL;
   HMI_FIT503.ALL := FIT503_FB.ALL;
   AIT504_FB : AIN_FBD(WRIO_Enb := DI_WIFI_RIO_5, Raw_RIO := AI_AIT_504_COND, Raw_WRIO := W_AI_AIT_504_COND, L_Raw_RIO := 0, H_Raw_RIO := 31208, L_Raw_WRIO := 3277, H_Raw_WRIO := 16383, HEU := 1200, LEU := 0.0, SAHH := HMI_AIT504.SAHH, SAH := HMI_AIT504.SAH, SAL := HMI_AIT504.SAL, SALL := HMI_AIT504.SALL, Simulation := HMI_AIT504.Sim, RIO_Hty := AI_AIT_504_COND_HTY, WRIO_Hty := W_AI_AIT_504_COND_HTY, HMI := HMI_AIT504, Pv := HMI_AIT504.Pv, Sim_PV := HMI_AIT504.Sim_PV);
   HMI_AIT504.Wifi_Enb := AIT504_FB.Wifi_Enb;
   HMI_AIT504.AHH := AIT504_FB.AHH;
   HMI_AIT504.ALL := AIT504_FB.ALL;
   HMI_AIT504.Hty := AIT504_FB.Hty;
   HMI_AIT504.AH := AIT504_FB.AH;
   HMI_AIT504.AL := AIT504_FB.AL;
   MV504_FB : MV_FBD(Auto := HMI_MV504.Auto, AutoInp := _MV504_AutoInp, ZSO := DI_MV_504_ZSO, Open_TM := 15, ZSC := DI_MV_504_ZSC, Close_TM := 15, Cmd := HMI_MV504.Cmd, HMI := HMI_MV504);
   FIT504_FB : FIT_FBD(WRIO_Enb := DI_WIFI_RIO_5, Raw_RIO := AI_FIT_504_FLOW, Raw_WRIO := W_AI_FIT_504_FLOW, L_Raw_RIO := -15, H_Raw_RIO := 31208, L_Raw_WRIO := 3277, H_Raw_WRIO := 16383, HEU := 2, LEU := 0.0, SAHH := HMI_FIT504.SAHH, SAH := HMI_FIT504.SAH, SAL := HMI_FIT504.SAL, SALL := HMI_FIT504.SALL, Simulation := HMI_FIT504.Sim, RIO_Hty := AI_FIT_504_FLOW_HTY, WRIO_Hty := W_AI_FIT_504_FLOW_HTY, Totaliser_Enb := _FIT504_Tot_Enb, Rst_Totaliser := HMI_FIT504.Rst_Totaliser, HMI := HMI_FIT504, Pv := HMI_FIT504.Pv, Sim_Pv := HMI_FIT504.Sim_PV, Totaliser := HMI_FIT504.Totaliser);
   DO_MV_504_CLOSE := MV504_FB.Cmd_Close;
   DO_MV_504_OPEN := MV504_FB.Cmd_Open;
   HMI_MV504.FTO := MV504_FB.FTO;
   HMI_MV504.FTC := MV504_FB.FTC;
   HMI_FIT504.Wifi_Enb := FIT504_FB.Wifi_Enb;
   HMI_FIT504.AHH := FIT504_FB.AHH;
   HMI_FIT504.Hty := FIT504_FB.Hty;
   HMI_FIT504.AH := FIT504_FB.AH;
   HMI_FIT504.AL := FIT504_FB.AL;
   HMI_FIT504.ALL := FIT504_FB.ALL;
   PSL501_FB : SWITCH_FBD(Alarm := DI_PSL_501_LOW, Delay := HMI_PSL501.Delay, HMI := HMI_PSL501);
   HMI_PSL501.Alarm := PSL501_FB.Status;
   PSH501_FB : SWITCH_FBD(Alarm := DI_PSH_501_HIGH, Delay := HMI_PSH501.Delay, HMI := HMI_PSH501);
   HMI_PSH501.Alarm := PSH501_FB.Status;
END_ROUTINE

ROUTINE IO   (* structured text *)
   (*DIGITAL INPUTS*)
   DI_WIFI_PLC_5	:=RIO5:0:I.Data.0;
   DI_WIFI_RIO_5	:=RIO5:0:I.Data.1;
   DI_P_501_AUTO	:=RIO5:0:I.Data.2;
   DI_P_501_FAULT	:=RIO5:0:I.Data.3;
   DI_P_501_RUN	:=RIO5:0:I.Data.4;
   DI_P_502_AUTO	:=RIO5:0:I.Data.5;
   DI_P_502_FAULT	:=RIO5:0:I.Data.6;
   DI_P_502_RUN	:=RIO5:0:I.Data.7;
   DI_MV_501_ZSO	:=RIO5:0:I.Data.8;
   DI_MV_501_ZSC	:=RIO5:0:I.Data.9;
   DI_MV_502_ZSO	:=RIO5:0:I.Data.10;
   DI_MV_502_ZSC	:=RIO5:0:I.Data.11;
   DI_MV_503_ZSO	:=RIO5:0:I.Data.12;
   DI_MV_503_ZSC	:=RIO5:0:I.Data.13;
   DI_MV_504_ZSO	:=RIO5:0:I.Data.14;
   DI_MV_504_ZSC	:=RIO5:0:I.Data.15;
   DI_PSL_501_LOW	:=RIO5:0:I.Data.16;
   DI_PSH_501_HIGH	:=RIO5:0:I.Data.17;
   DI_VSD_1_PB		:=RIO5:0:I.Data.18;
   DI_VSD_2_PB		:=RIO5:0:I.Data.19;
   DI_RIO5_SPARE_20:=RIO5:0:I.Data.20;
   DI_RIO5_SPARE_21:=RIO5:0:I.Data.21;
   DI_RIO5_SPARE_22:=RIO5:0:I.Data.22;
   DI_RIO5_SPARE_23:=RIO5:0:I.Data.23;
   DI_RIO5_SPARE_24:=RIO5:0:I.Data.24;
   DI_RIO5_SPARE_25:=RIO5:0:I.Data.25;
   DI_RIO5_SPARE_26:=RIO5:0:I.Data.26;
   DI_RIO5_SPARE_27:=RIO5:0:I.Data.27;
   DI_RIO5_SPARE_28:=RIO5:0:I.Data.28;
   DI_RIO5_SPARE_29:=RIO5:0:I.Data.29;
   DI_RIO5_SPARE_30:=RIO5:0:I.Data.30;
   DI_RIO5_SPARE_31:=RIO5:0:I.Data.31;
   
   (*DIGITAL OUTPUTS*)
   RIO5:1:O.0	:=DO_MV_501_OPEN;
   RIO5:1:O.1	:=DO_MV_501_CLOSE;
   RIO5:1:O.2	:=DO_MV_502_OPEN;
   RIO5:1:O.3	:=DO_MV_502_CLOSE;
   RIO5:1:O.4	:=DO_MV_503_OPEN;
   RIO5:1:O.5	:=DO_MV_503_CLOSE;
   RIO5:1:O.6	:=DO_MV_504_OPEN;
   RIO5:1:O.7	:=DO_MV_504_CLOSE;
   RIO5:1:O.8	:=DO_RIO5_SPARE_08;
   RIO5:1:O.9	:=DO_RIO5_SPARE_09;
   RIO5:1:O.10	:=DO_LED_RED;
   RIO5:1:O.11	:=DO_RIO5_SPARE_11;
   RIO5:1:O.12	:=DO_RIO5_SPARE_12;
   RIO5:1:O.13	:=DO_RIO5_SPARE_13;
   RIO5:1:O.14	:=DO_RIO5_SPARE_14;
   RIO5:1:O.15	:=DO_RIO5_SPARE_15;
   
   (*ANALOG INPUTS*)
   AI_AIT_501_PH		:=RIO5:2:I.Ch0Data;
   AI_AIT_502_ORP		:=RIO5:2:I.Ch1Data;
   AI_AIT_503_COND		:=RIO5:2:I.Ch2Data;
   AI_AIT_504_COND		:=RIO5:2:I.Ch3Data;
   AI_FIT_501_FLOW		:=RIO5:2:I.Ch4Data;
   AI_FIT_502_FLOW		:=RIO5:2:I.Ch5Data;
   AI_FIT_503_FLOW		:=RIO5:2:I.Ch6Data;
   AI_FIT_504_FLOW		:=RIO5:2:I.Ch7Data;
   AI_PIT_501_PRESS	:=RIO5:2:I.Ch8Data;
   AI_PIT_502_PRESS	:=RIO5:2:I.Ch9Data;
   AI_PIT_503_PRESS	:=RIO5:2:I.Ch10Data;
   AI_RIO5_SPARE_11	:=RIO5:2:I.Ch11Data;
   
   AI_AIT_501_PH_HTY		:=(NOT RIO5:2:I.GeneralFault);
   AI_AIT_502_ORP_HTY		:=(NOT RIO5:2:I.GeneralFault);
   AI_AIT_503_COND_HTY		:=(NOT RIO5:2:I.GeneralFault);
   AI_AIT_504_COND_HTY		:=(NOT RIO5:2:I.GeneralFault);
   AI_FIT_501_FLOW_HTY		:=(NOT RIO5:2:I.GeneralFault);
   AI_FIT_502_FLOW_HTY		:=(NOT RIO5:2:I.GeneralFault);
   AI_FIT_503_FLOW_HTY		:=(NOT RIO5:2:I.GeneralFault);
   AI_FIT_504_FLOW_HTY		:=(NOT RIO5:2:I.GeneralFault);
   AI_PIT_501_PRESS_HTY	:=(NOT RIO5:2:I.GeneralFault);
   AI_PIT_502_PRESS_HTY	:=(NOT RIO5:2:I.GeneralFault);
   AI_PIT_503_PRESS_HTY	:=(NOT RIO5:2:I.GeneralFault);
   AI_RIO4_SPARE_11_HTY	:=(NOT RIO5:2:I.GeneralFault);
   
   (*WIRELESS ANALOG INPUTS*)
   W_AI_AIT_501_PH		:=WRIO5:1:I.Ch0Data;
   W_AI_AIT_502_ORP	:=WRIO5:1:I.Ch1Data;
   W_AI_AIT_503_COND	:=WRIO5:1:I.Ch2Data;
   W_AI_AIT_504_COND	:=WRIO5:1:I.Ch3Data;
   W_AI_FIT_501_FLOW	:=WRIO5:1:I.Ch4Data;
   W_AI_FIT_502_FLOW	:=WRIO5:1:I.Ch5Data;
   W_AI_FIT_503_FLOW	:=WRIO5:1:I.Ch6Data;
   W_AI_FIT_504_FLOW	:=WRIO5:1:I.Ch7Data;
   W_AI_PIT_501_PRESS	:=WRIO5:2:I.Ch0Data;
   W_AI_PIT_502_PRESS	:=WRIO5:2:I.Ch1Data;
   W_AI_PIT_503_PRESS	:=WRIO5:2:I.Ch2Data;
   
   W_AI_AIT_501_PH_HTY		:=WRIO5:1:I.Ch0Fault ;
   W_AI_AIT_502_ORP_HTY	:=WRIO5:1:I.Ch1Fault ;
   W_AI_AIT_503_COND_HTY	:=WRIO5:1:I.Ch2Fault ;
   W_AI_AIT_504_COND_HTY	:=WRIO5:1:I.Ch3Fault ;
   W_AI_FIT_501_FLOW_HTY	:=WRIO5:1:I.Ch4Fault ;
   W_AI_FIT_502_FLOW_HTY	:=WRIO5:1:I.Ch5Fault ;
   W_AI_FIT_503_FLOW_HTY	:=WRIO5:1:I.Ch6Fault ;
   W_AI_FIT_504_FLOW_HTY	:=WRIO5:1:I.Ch7Fault ;
   
   W_AI_PIT_501_PRESS_HTY	:=WRIO5:2:I.Ch0Fault ;
   W_AI_PIT_502_PRESS_HTY	:=WRIO5:2:I.Ch1Fault ;
   W_AI_PIT_503_PRESS_HTY	:=WRIO5:2:I.Ch2Fault ;
   
   (*Wireless Selction*)
   HMI_WIFI.PLC_WIFI		:= DI_WIFI_PLC_5;
   HMI_WIFI.RIO_WIFI		:= DI_WIFI_RIO_5;
   
   
   
END_ROUTINE

ROUTINE Logix_Status   (* ladder *)
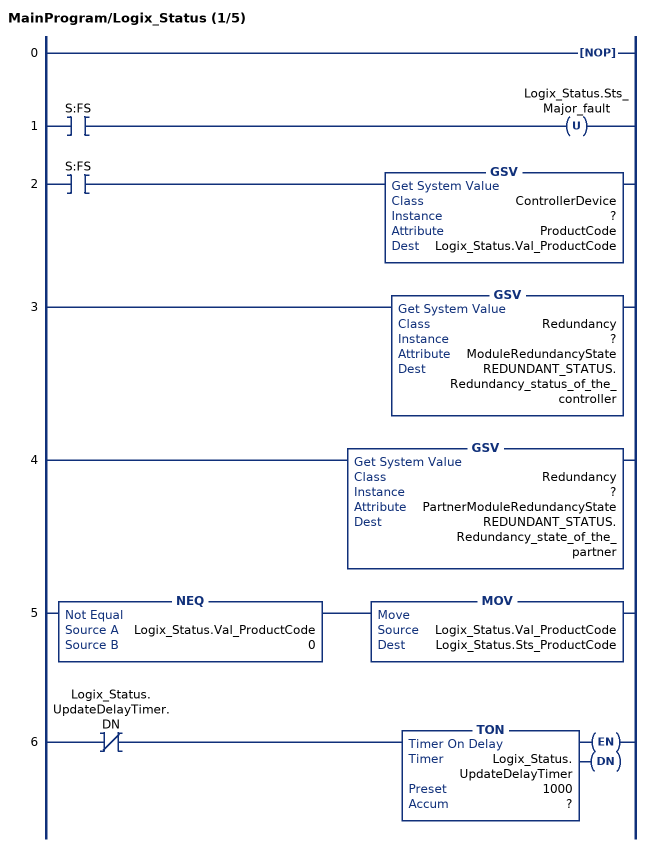
   0: NOP();
   1: XIC(S:FS)OTU(Logix_Status.Sts_Major_fault);
   2: XIC(S:FS)GSV(ControllerDevice,?,ProductCode,Logix_Status.Val_ProductCode);
   3: GSV(Redundancy,?,ModuleRedundancyState,REDUNDANT_STATUS.Redundancy_status_of_the_controller);
   4: GSV(Redundancy,?,PartnerModuleRedundancyState,REDUNDANT_STATUS.Redundancy_state_of_the_partner);
   5: NEQ(Logix_Status.Val_ProductCode,0)MOV(Logix_Status.Val_ProductCode,Logix_Status.Sts_ProductCode);
   6: XIO(Logix_Status.UpdateDelayTimer.DN)TON(Logix_Status.UpdateDelayTimer,?,?);
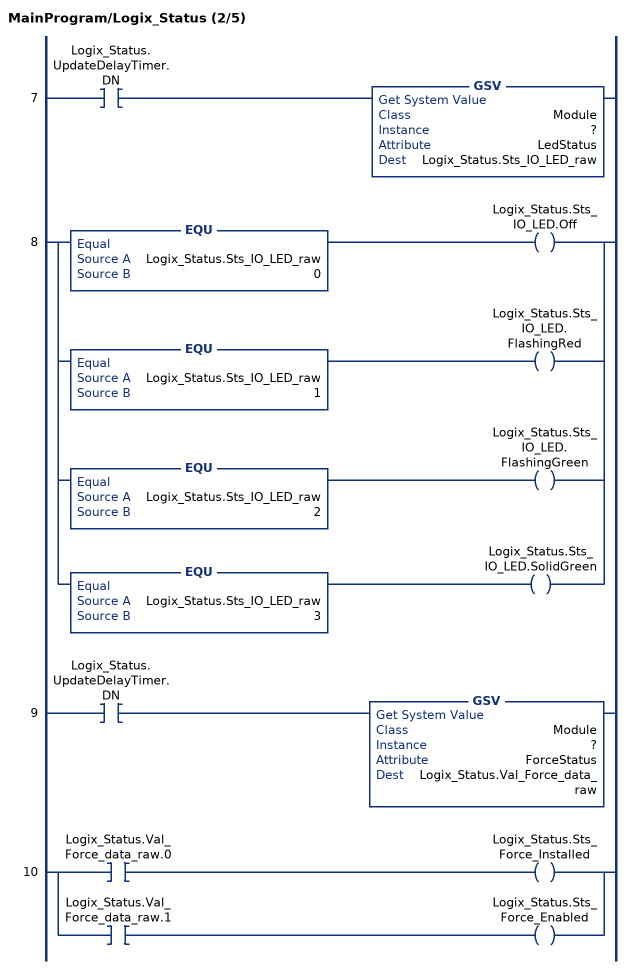
   7: XIC(Logix_Status.UpdateDelayTimer.DN)GSV(Module,?,LedStatus,Logix_Status.Sts_IO_LED_raw);
   8: [EQU(Logix_Status.Sts_IO_LED_raw,0) OTE(Logix_Status.Sts_IO_LED.Off) ,EQU(Logix_Status.Sts_IO_LED_raw,1) OTE(Logix_Status.Sts_IO_LED.FlashingRed) ,EQU(Logix_Status.Sts_IO_LED_raw,2) OTE(Logix_Status.Sts_IO_LED.FlashingGreen) ,EQU(Logix_Status.Sts_IO_LED_raw,3) OTE(Logix_Status.Sts_IO_LED.SolidGreen) ];
   9: XIC(Logix_Status.UpdateDelayTimer.DN)GSV(Module,?,ForceStatus,Logix_Status.Val_Force_data_raw);
   10: [XIC(Logix_Status.Val_Force_data_raw.0) OTE(Logix_Status.Sts_Force_Installed) ,XIC(Logix_Status.Val_Force_data_raw.1) OTE(Logix_Status.Sts_Force_Enabled) ];
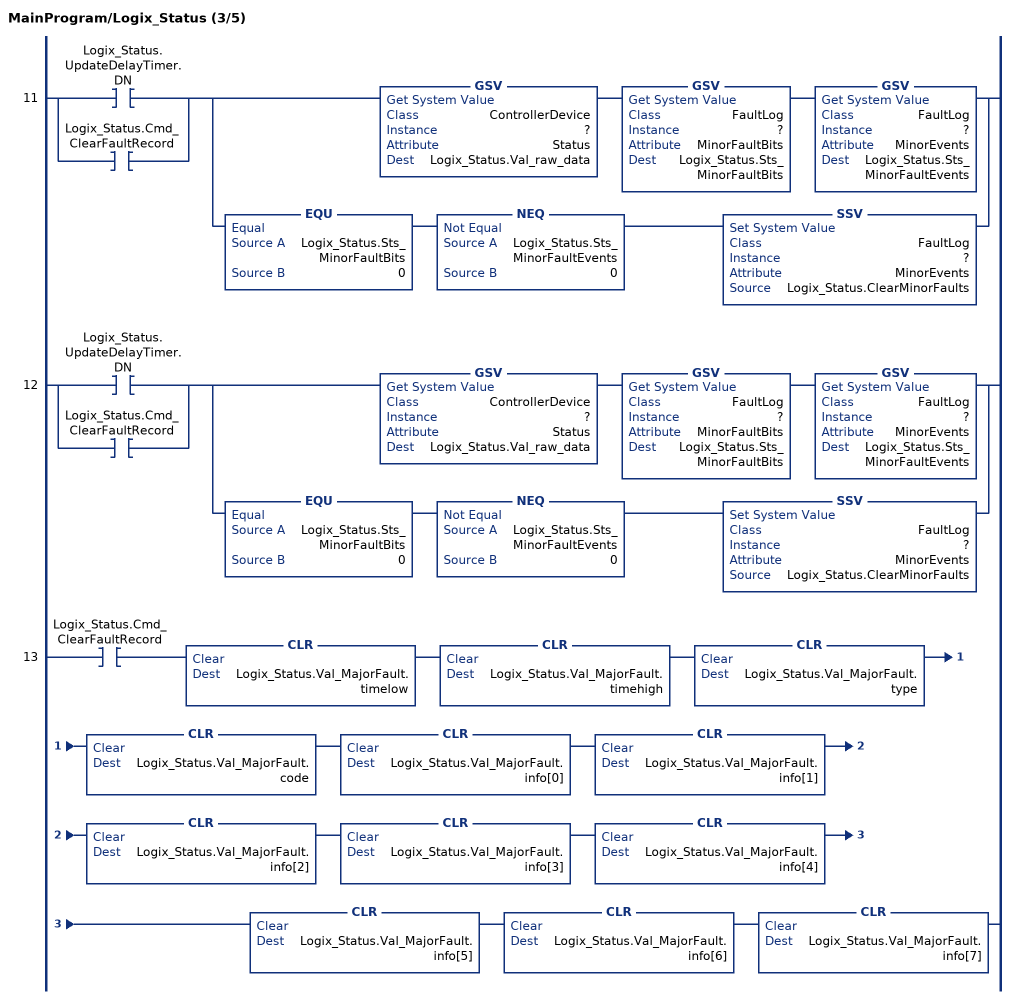
   11: [XIC(Logix_Status.UpdateDelayTimer.DN) ,XIC(Logix_Status.Cmd_ClearFaultRecord) ][GSV(ControllerDevice,?,Status,Logix_Status.Val_raw_data) GSV(FaultLog,?,MinorFaultBits,Logix_Status.Sts_MinorFaultBits) GSV(FaultLog,?,MinorEvents,Logix_Status.Sts_MinorFaultEvents) ,EQU(Logix_Status.Sts_MinorFaultBits,0) NEQ(Logix_Status.Sts_MinorFaultEvents,0) SSV(FaultLog,?,MinorEvents,Logix_Status.ClearMinorFaults) ];
   12: [XIC(Logix_Status.UpdateDelayTimer.DN) ,XIC(Logix_Status.Cmd_ClearFaultRecord) ][GSV(ControllerDevice,?,Status,Logix_Status.Val_raw_data) GSV(FaultLog,?,MinorFaultBits,Logix_Status.Sts_MinorFaultBits) GSV(FaultLog,?,MinorEvents,Logix_Status.Sts_MinorFaultEvents) ,EQU(Logix_Status.Sts_MinorFaultBits,0) NEQ(Logix_Status.Sts_MinorFaultEvents,0) SSV(FaultLog,?,MinorEvents,Logix_Status.ClearMinorFaults) ];
   13: XIC(Logix_Status.Cmd_ClearFaultRecord)CLR(Logix_Status.Val_MajorFault.timelow)CLR(Logix_Status.Val_MajorFault.timehigh)CLR(Logix_Status.Val_MajorFault.type)CLR(Logix_Status.Val_MajorFault.code)CLR(Logix_Status.Val_MajorFault.info[0])CLR(Logix_Status.Val_MajorFault.info[1])CLR(Logix_Status.Val_MajorFault.info[2])CLR(Logix_Status.Val_MajorFault.info[3])CLR(Logix_Status.Val_MajorFault.info[4])CLR(Logix_Status.Val_MajorFault.info[5])CLR(Logix_Status.Val_MajorFault.info[6])CLR(Logix_Status.Val_MajorFault.info[7]);
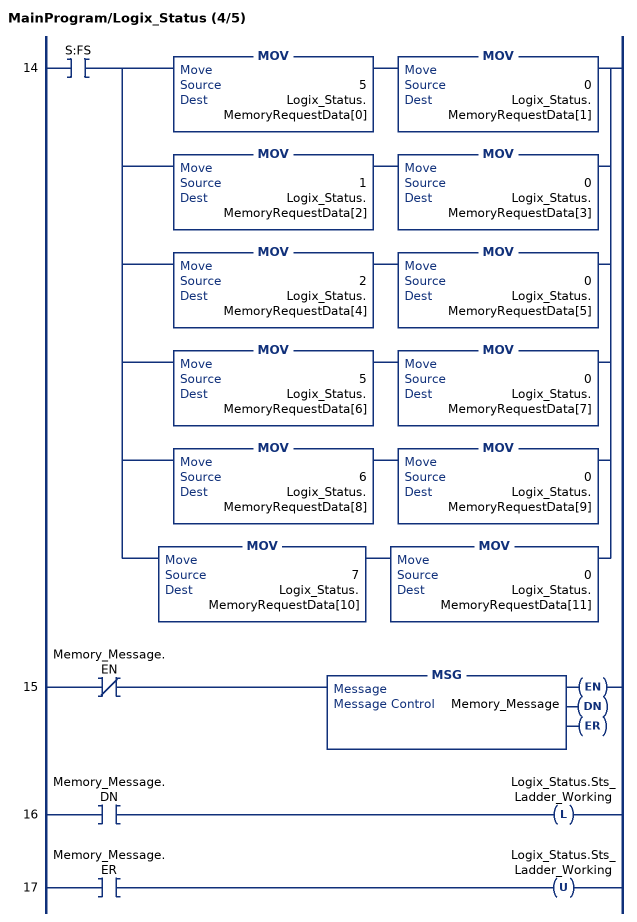
   14: XIC(S:FS)[MOV(5,Logix_Status.MemoryRequestData[0]) MOV(0,Logix_Status.MemoryRequestData[1]) ,MOV(1,Logix_Status.MemoryRequestData[2]) MOV(0,Logix_Status.MemoryRequestData[3]) ,MOV(2,Logix_Status.MemoryRequestData[4]) MOV(0,Logix_Status.MemoryRequestData[5]) ,MOV(5,Logix_Status.MemoryRequestData[6]) MOV(0,Logix_Status.MemoryRequestData[7]) ,MOV(6,Logix_Status.MemoryRequestData[8]) MOV(0,Logix_Status.MemoryRequestData[9]) ,MOV(7,Logix_Status.MemoryRequestData[10]) MOV(0,Logix_Status.MemoryRequestData[11]) ];
   15: XIO(Memory_Message.EN)MSG(Memory_Message);
   16: XIC(Memory_Message.DN)OTL(Logix_Status.Sts_Ladder_Working);
   17: XIC(Memory_Message.ER)OTU(Logix_Status.Sts_Ladder_Working);
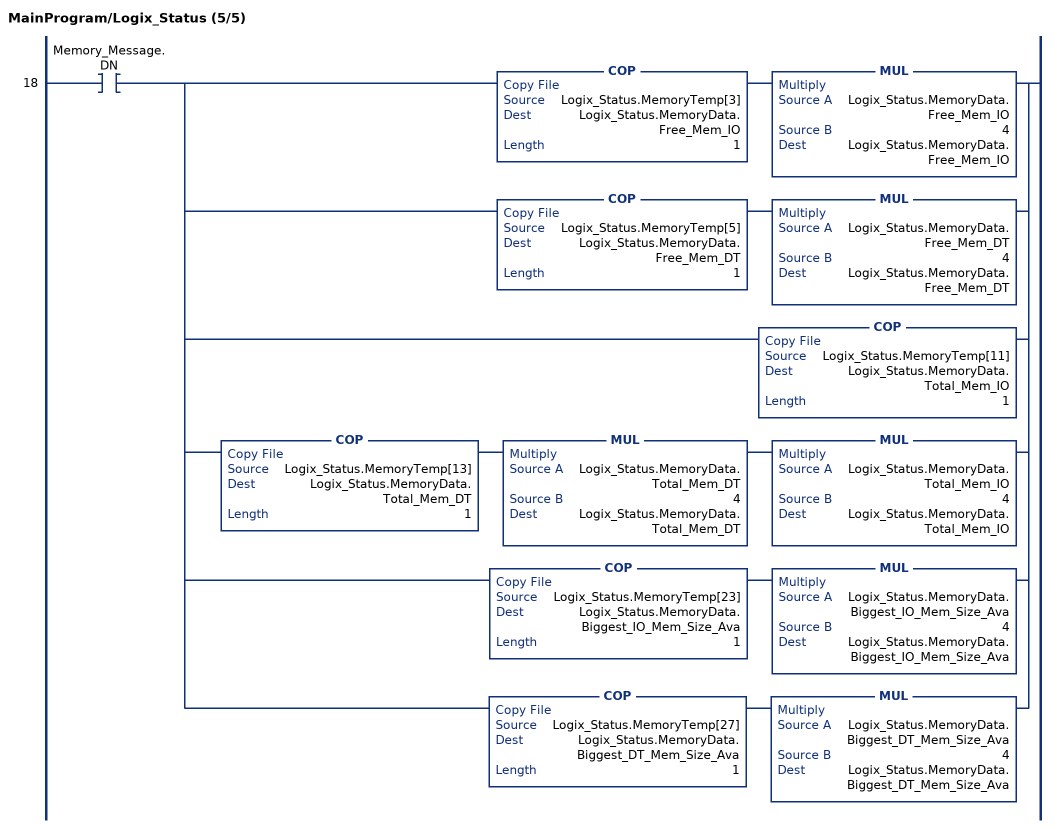
   18: XIC(Memory_Message.DN)[COP(Logix_Status.MemoryTemp[3],Logix_Status.MemoryData.Free_Mem_IO,1) MUL(Logix_Status.MemoryData.Free_Mem_IO,4,Logix_Status.MemoryData.Free_Mem_IO) ,COP(Logix_Status.MemoryTemp[5],Logix_Status.MemoryData.Free_Mem_DT,1) MUL(Logix_Status.MemoryData.Free_Mem_DT,4,Logix_Status.MemoryData.Free_Mem_DT) ,COP(Logix_Status.MemoryTemp[11],Logix_Status.MemoryData.Total_Mem_IO,1) ,COP(Logix_Status.MemoryTemp[13],Logix_Status.MemoryData.Total_Mem_DT,1) MUL(Logix_Status.MemoryData.Total_Mem_DT,4,Logix_Status.MemoryData.Total_Mem_DT) MUL(Logix_Status.MemoryData.Total_Mem_IO,4,Logix_Status.MemoryData.Total_Mem_IO) ,COP(Logix_Status.MemoryTemp[23],Logix_Status.MemoryData.Biggest_IO_Mem_Size_Ava,1) MUL(Logix_Status.MemoryData.Biggest_IO_Mem_Size_Ava,4,Logix_Status.MemoryData.Biggest_IO_Mem_Size_Ava) ,COP(Logix_Status.MemoryTemp[27],Logix_Status.MemoryData.Biggest_DT_Mem_Size_Ava,1) MUL(Logix_Status.MemoryData.Biggest_DT_Mem_Size_Ava,4,Logix_Status.MemoryData.Biggest_DT_Mem_Size_Ava) ];
END_ROUTINE

ROUTINE Main_Seq   (* structured text *)
   
   (*SECOND PULSE*)
   TON.PRE	:=1000;
   TON.TimerEnable	:=1;
   TONR(TON );
   R_TRIG.InputBit :=TON.DN ;
   OSRI( R_TRIG);
   _SEC_P  := R_TRIG.OutputBit;
   TON.Reset := _SEC_P;
   
   IF HMI_PLANT.STOP THEN
   	HMI_P5_STATE:=13;
   END_IF;
   
   (*
   IF HMI_SHUTDOWN_FLUSHING.ON AND HMI_P5_SD_FLUSHING_DONE.ON THEN
   	HMI_P5_STATE:=19;
   END_IF ;
   *)
   
   (*
   if S:FS then
   	HMI_P5_STATE := 1;
   end_if;
   *)
   
   
   HMI_RO_TMP	:=((HMI_PIT501.PV+ HMI_PIT503.PV)/2)-HMI_PIT502.PV ;
   
   
   
   (*MINUTES PULSE*)
   TON_MIN.PRE	 :=60000;
   TON_MIN.TimerEnable	:=1;
   TONR(TON_MIN );
   R_TRIG_MIN.InputBit :=TON_MIN.DN ;
   OSRI( R_TRIG_MIN);
   _MIN_P  := R_TRIG_MIN.OutputBit;
   TON_MIN.Reset := _MIN_P;
   
   IF _SEC_P THEN
   	_SEC_TEST:=_SEC_TEST+1;
   END_IF;
   
   IF _MIN_P THEN
   	TEST_MIN:=TEST_MIN+1;
   END_IF;
   
   HMI_HPP_Q_MAX_M3H	 		:= 2;
   HMI_HPP_Q_SET_M3H 			:= 0.6;
   HMI_MIN_RO_VSD_SPEED		:= HMI_HPP_Q_SET_M3H/ HMI_HPP_Q_MAX_M3H *50 *0.1;
   HMI_RAMPING_RATE_PER_SEC	:= 1.5 ;(*HMI_HPP_Q_SET_M3H *0.025 *50;*)
   HMI_VSD_MIN_SPEED			:= 10;
   (*HMI_VSD_HIGH_SPEED			:= 27;*)
   HMI_VSD_HIGH_SPEED			:= 30;
   
   (*-----------WRITE FAULT CONDITION--------------*)
   
   CASE HMI_P5_STATE OF
   	1:(*PLANT IN STANDBY*)
   		_P_RO_HIGH_AutoInp		:= 0;
   		_MV501_AutoInp			:= 0;
   		_MV502_AutoInp			:= 0;
   		_MV503_AutoInp			:= 0;
   		_MV504_AutoInp			:= 0;
   		_P50X_AutoSpeed			:= HMI_VSD_MIN_SPEED;
   
   		HMI_RO_HPP_SD.ON			:=0;
   		HMI_FLUSHING_MIN			:=0;
   		HMI_RO_SD_FLUSHING_MIN		:=0;
   		HMI_RO_HIGH_PUMP_SHUTDOWN	:=0;
   		HMI_P5_SD_FLUSHING_DONE.ON	:=0;
   		HMI_MV501_TIMEOUT_TM		:=0;
   		HMI_MV502_TIMEOUT_TM		:=0;
   		HMI_MV503_TIMEOUT_TM		:=0;
   		HMI_MV504_TIMEOUT_TM		:=0;
   
   		IF HMI_P5_PERMISSIVE.ON AND HMI_PLANT.START THEN
   			_NEXT:=0;
   			HMI_P5_STATE:=3;
   		END_IF;
   
   	2:(*CHECK RO FEED PUMP STATUS*)
   		_P_RO_HIGH_AutoInp	:= 0;
   		_MV501_AutoInp		:= 0;
   		_MV502_AutoInp		:= 0;
   		_MV503_AutoInp		:= 0;
   		_MV504_AutoInp		:= 0;
   		_P50X_AutoSpeed		:= HMI_VSD_MIN_SPEED;
   
   		HMI_RO_HPP_SD.ON			:=0;
   		HMI_FLUSHING_MIN			:=0;
   		HMI_RO_SD_FLUSHING_MIN		:=0;
   		HMI_RO_HIGH_PUMP_SHUTDOWN	:=0;
   		HMI_P5_SD_FLUSHING_DONE.ON	:=0;
   		HMI_MV501_TIMEOUT_TM		:=0;
   		HMI_MV502_TIMEOUT_TM		:=0;
   		HMI_MV503_TIMEOUT_TM		:=0;
   		HMI_MV504_TIMEOUT_TM		:=0;
   
   		IF HMI_P_RO_FEED_DUTY.Pump_Running AND _NEXT THEN
   			_NEXT:=0;
   			HMI_P5_STATE:=3;
   		END_IF;
   
   	3:(*OPEN MV503, 504 , OPEN UF BACKWASH VALVE , DRAIN VALVE *)
   	   	_P_RO_HIGH_AutoInp	:= 0;
   		_MV501_AutoInp		:= 0;
   	 	_MV502_AutoInp		:= 0;
   		_MV503_AutoInp		:= 1;
   		_MV504_AutoInp		:= 1;
   		_P50X_AutoSpeed		:= HMI_VSD_MIN_SPEED;
   
   		HMI_RO_HPP_SD.ON			:=0;
   		HMI_FLUSHING_MIN			:=0;
   		HMI_RO_SD_FLUSHING_MIN		:=0;
   		HMI_RO_HIGH_PUMP_SHUTDOWN	:=0;
   		HMI_P5_SD_FLUSHING_DONE.ON	:=0;
   		HMI_MV501_TIMEOUT_TM		:=0;
   		HMI_MV502_TIMEOUT_TM		:=0;
   		HMI_MV503_TIMEOUT_TM		:=0;
   		HMI_MV504_TIMEOUT_TM		:=0;
   
   		IF HMI_MV503.STATUS=2 AND HMI_MV504.STATUS=2 AND HMI_P_RO_FEED_DUTY.Pump_Running OR _NEXT THEN
   			_NEXT:=0;
   			HMI_P5_STATE:=4;
   		END_IF;
   
   	4:(*LOW PRESSURE FLUSHING *)
   		_P_RO_HIGH_AutoInp	:= 0;
   		_MV501_AutoInp		:= 0;
   		_MV502_AutoInp		:= 0;
   		_MV503_AutoInp		:= 1;
   		_MV504_AutoInp		:= 1;
   		_P50X_AutoSpeed		:= HMI_VSD_MIN_SPEED;
   
   		HMI_RO_HPP_SD.ON			:=0;
   		HMI_RO_SD_FLUSHING_MIN		:=0;
   		HMI_RO_HIGH_PUMP_SHUTDOWN	:=0;
   		HMI_MV501_TIMEOUT_TM		:=0;
   		HMI_MV502_TIMEOUT_TM		:=0;
   		HMI_MV503_TIMEOUT_TM		:=0;
   		HMI_MV504_TIMEOUT_TM		:=0;
   
   		IF _MIN_P THEN
   			HMI_FLUSHING_MIN:= HMI_FLUSHING_MIN+1;
   		END_IF;
   
   
   
   
   		IF HMI_FLUSHING_MIN>HMI_FLUSHING_MIN_SP OR _NEXT THEN
   			HMI_P5_SD_FLUSHING_DONE.ON	:=1;
   			_NEXT :=0;
   			HMI_P5_STATE:=5;
   
   		END_IF;
   
   	5:(*START HIGH PRESSURE PUMP , FREQUENCY EQUAL TO 10% OF TARGET FLOW RATE   *)
   		_P_RO_HIGH_AutoInp	:= 1;
   		_MV501_AutoInp		:= 0;
   		_MV502_AutoInp		:= 0;
   		_MV503_AutoInp		:= 1;
   		_MV504_AutoInp		:= 1;
   		_P50X_AutoSpeed		:= HMI_VSD_MIN_SPEED;
   
   		HMI_RO_HPP_SD.ON			:=0;
   		HMI_FLUSHING_MIN			:=0;
   		HMI_RO_SD_FLUSHING_MIN		:=0;
   		HMI_RO_HIGH_PUMP_SHUTDOWN	:=0;
   		HMI_P5_SD_FLUSHING_DONE.ON	:=0;
   		HMI_MV501_TIMEOUT_TM		:=0;
   		HMI_MV502_TIMEOUT_TM		:=0;
   		HMI_MV503_TIMEOUT_TM		:=0;
   		HMI_MV504_TIMEOUT_TM		:=0;
   
   		IF (HMI_P501.Speed >= _P50X_AutoSpeed) OR (HMI_P502.Speed >= _P50X_AutoSpeed) OR _NEXT THEN
   			_NEXT:=0;
   			HMI_P5_STATE:=6;
   		END_IF;
   
   	6:(*MAINTAIN AT LEAST 10% OF FIT501 FLOW , RAMP 4.5 /SEC OF FINAL FLOW UNTIL REACH DESIRED FLOW *)
   		_P_RO_HIGH_AutoInp	:= 1;
   		_MV501_AutoInp		:= 0;
   		_MV502_AutoInp		:= 0;
   		_MV503_AutoInp		:= 1;
   		_MV504_AutoInp		:= 1;
   
   		HMI_RO_HPP_SD.ON			:=0;
   		HMI_FLUSHING_MIN			:=0;
   		HMI_RO_SD_FLUSHING_MIN		:=0;
   		HMI_RO_HIGH_PUMP_SHUTDOWN	:=0;
   		HMI_P5_SD_FLUSHING_DONE.ON	:=0;
   		HMI_MV501_TIMEOUT_TM		:=0;
   		HMI_MV502_TIMEOUT_TM		:=0;
   		HMI_MV503_TIMEOUT_TM		:=0;
   		HMI_MV504_TIMEOUT_TM		:=0;
   
   		IF  _P50X_AutoSpeed <  HMI_VSD_HIGH_SPEED   THEN
   			IF _SEC_P THEN
   				IF (*((HMI_FIT503.PV/HMI_FIT501.PV)< 0.3) AND *)(HMI_PIT502.PV<HMI_PIT503.PV) AND HMI_PIT501.PV<275 THEN
   					_P50X_AutoSpeed :=  _P50X_AutoSpeed + 0.5 ;
   				END_IF;
   			END_IF;
   		END_IF;
   
   		 (*IF ((HMI_FIT501.Pv > HMI_HPP_Q_SET_M3H) AND (HMI_PIT502.PV<HMI_PIT503.PV)) AND HMI_PIT501.PV>250 OR _NEXT THEN *)
           IF ((HMI_FIT501.Pv > HMI_HPP_Q_SET_M3H) AND (HMI_PIT502.PV<HMI_PIT503.PV) AND (HMI_PIT501.PV>260)) THEN
   				_NEXT:=0;
   				HMI_P5_STATE:=7;
   		END_IF;
   
   
   	7:(*CHECK CONDUCTIVITY > CONDUCTIVITY SETPOINT *)
   		_P_RO_HIGH_AutoInp	:= 1;
   		_MV501_AutoInp		:= 0;
   		_MV502_AutoInp		:= 0;
   		_MV503_AutoInp		:= 1;
   		_MV504_AutoInp		:= 1;
   
   		HMI_RO_HPP_SD.ON			:=0;
   		HMI_FLUSHING_MIN			:=0;
   		HMI_RO_SD_FLUSHING_MIN		:=0;
   		HMI_RO_HIGH_PUMP_SHUTDOWN	:=0;
   		HMI_P5_SD_FLUSHING_DONE.ON	:=0;
   		HMI_MV501_TIMEOUT_TM		:=0;
   		HMI_MV502_TIMEOUT_TM		:=0;
   		HMI_MV503_TIMEOUT_TM		:=0;
   		HMI_MV504_TIMEOUT_TM		:=0;
   
   		IF HMI_AIT504.PV < HMI_AIT504.SAH OR _NEXT THEN
   			_NEXT:=0;
   			HMI_P5_STATE:=8;
   		END_IF;
   
   	8:(*OPEN MV501 PERMEATE VALVE  *)
   		_P_RO_HIGH_AutoInp	:= 1;
   		_MV501_AutoInp		:= 1;
   		_MV502_AutoInp		:= 0;
   		_MV503_AutoInp		:= 1;
   		_MV504_AutoInp		:= 1;
   
   		HMI_RO_HPP_SD.ON			:=0;
   		HMI_FLUSHING_MIN			:=0;
   		HMI_RO_SD_FLUSHING_MIN		:=0;
   		HMI_RO_HIGH_PUMP_SHUTDOWN	:=0;
   		HMI_P5_SD_FLUSHING_DONE.ON	:=0;
   		HMI_MV501_TIMEOUT_TM		:=0;
   		HMI_MV502_TIMEOUT_TM		:=0;
   		HMI_MV503_TIMEOUT_TM		:=0;
   		HMI_MV504_TIMEOUT_TM		:=0;
   
   		IF HMI_MV501.STATUS=2 OR _NEXT THEN
   			_NEXT:=0;
   			HMI_P5_STATE:=9;
   		END_IF;
   
   	9:(*CLOSE MV503   *)
   		_P_RO_HIGH_AutoInp	:= 1;
   		_MV501_AutoInp		:= 1;
   		_MV502_AutoInp		:= 0;
   		_MV503_AutoInp		:= 0;
   		_MV504_AutoInp		:= 1;
   
   		HMI_RO_HPP_SD.ON			:=0;
   		HMI_FLUSHING_MIN			:=0;
   		HMI_RO_SD_FLUSHING_MIN		:=0;
   		HMI_RO_HIGH_PUMP_SHUTDOWN	:=0;
   		HMI_P5_SD_FLUSHING_DONE.ON	:=0;
   		HMI_MV501_TIMEOUT_TM		:=0;
   		HMI_MV502_TIMEOUT_TM		:=0;
   		HMI_MV503_TIMEOUT_TM		:=0;
   		HMI_MV504_TIMEOUT_TM		:=0;
   
   		IF HMI_MV503.STATUS=1 OR _NEXT THEN
   			_NEXT:=0;
   			HMI_P5_STATE:=10;
   		END_IF;
   
   	10:(*OPEN MV502   *)
   		_P_RO_HIGH_AutoInp	:= 1;
   		_MV501_AutoInp		:= 1;
   		_MV502_AutoInp		:= 1;
   		_MV503_AutoInp		:= 0;
   		_MV504_AutoInp		:= 1;
   
   		HMI_RO_HPP_SD.ON			:=0;
   		HMI_FLUSHING_MIN			:=0;
   		HMI_RO_SD_FLUSHING_MIN		:=0;
   		HMI_RO_HIGH_PUMP_SHUTDOWN	:=0;
   		HMI_P5_SD_FLUSHING_DONE.ON	:=0;
   		HMI_MV501_TIMEOUT_TM		:=0;
   		HMI_MV502_TIMEOUT_TM		:=0;
   		HMI_MV503_TIMEOUT_TM		:=0;
   		HMI_MV504_TIMEOUT_TM		:=0;
   
   
   		IF HMI_MV502.STATUS=2 OR _NEXT THEN
   			_NEXT:=0;
   			HMI_P5_STATE:=11;
   		END_IF;
   
   	11:(*CLOSE MV504   *)
   		_P_RO_HIGH_AutoInp	:= 1;
   		_MV501_AutoInp		:= 1;
   		_MV502_AutoInp		:= 1;
   		_MV503_AutoInp		:= 0;
   		_MV504_AutoInp		:= 0;
   
   		HMI_RO_HPP_SD.ON			:=0;
   		HMI_FLUSHING_MIN			:=0;
   		HMI_RO_SD_FLUSHING_MIN		:=0;
   		HMI_RO_HIGH_PUMP_SHUTDOWN	:=0;
   		HMI_P5_SD_FLUSHING_DONE.ON	:=0;
   		HMI_MV501_TIMEOUT_TM		:=0;
   		HMI_MV502_TIMEOUT_TM		:=0;
   		HMI_MV503_TIMEOUT_TM		:=0;
   		HMI_MV504_TIMEOUT_TM		:=0;
   
   
   		IF HMI_MV504.STATUS=1 OR _NEXT THEN
   			_NEXT:=0;
   			HMI_P5_STATE:=12;
   		END_IF;
   
   	12:(*RO PERMEATE PRODUCTION*)
   		_P_RO_HIGH_AutoInp	:= 1;
   		_MV501_AutoInp		:= 1;
   		_MV502_AutoInp		:= 1;
   		_MV503_AutoInp		:= 0;
   		_MV504_AutoInp		:= 0;
   
   		HMI_RO_HPP_SD.ON			:=0;
   		HMI_FLUSHING_MIN			:=0;
   		HMI_RO_SD_FLUSHING_MIN		:=0;
   		HMI_RO_HIGH_PUMP_SHUTDOWN	:=0;
   		HMI_P5_SD_FLUSHING_DONE.ON	:=0;
   		HMI_MV501_TIMEOUT_TM		:=0;
   		HMI_MV502_TIMEOUT_TM		:=0;
   		HMI_MV503_TIMEOUT_TM		:=0;
   		HMI_MV504_TIMEOUT_TM		:=0;
   
   
   		IF HMI_PLANT.STOP OR _STOP  THEN
   			_STOP:=0;
   			HMI_P5_STATE:=13;
   		END_IF;
   
   	13:(*RAMP DOWN VSD*)
   		_P_RO_HIGH_AutoInp	:= 1;
   		_MV501_AutoInp		:= 1;
   		_MV502_AutoInp		:= 1;
   		_MV503_AutoInp		:= 0;
   		_MV504_AutoInp		:= 0;
   
   		HMI_RO_HPP_SD.ON			:=0;
   		HMI_FLUSHING_MIN			:=0;
   		HMI_RO_SD_FLUSHING_MIN		:=0;
   		HMI_RO_HIGH_PUMP_SHUTDOWN	:=0;
   		HMI_P5_SD_FLUSHING_DONE.ON	:=0;
   		HMI_MV501_TIMEOUT_TM		:=0;
   		HMI_MV502_TIMEOUT_TM		:=0;
   		HMI_MV503_TIMEOUT_TM		:=0;
   		HMI_MV504_TIMEOUT_TM		:=0;
   
   
   		IF  _P50X_AutoSpeed >  HMI_VSD_MIN_SPEED   THEN
   			IF _SEC_P THEN
   					_P50X_AutoSpeed :=  _P50X_AutoSpeed - 0.5 (*HMI_RAMPING_RATE_PER_SEC*) ;
   			END_IF;
   		END_IF;
   
   		IF  (HMI_P501.Speed <= HMI_VSD_MIN_SPEED) AND  (HMI_P502.Speed <= HMI_VSD_MIN_SPEED) OR _NEXT THEN
   			_NEXT:=0;
   			HMI_P5_STATE:=14;
   		END_IF;
   
   	14:(*STOP HPP*)
   		_P_RO_HIGH_AutoInp	:= 0;
   		_MV501_AutoInp		:= 1;
   		_MV502_AutoInp		:= 1;
   		_MV503_AutoInp		:= 0;
   		_MV504_AutoInp		:= 0;
   
   		HMI_RO_HPP_SD.ON			:=0;
   		HMI_FLUSHING_MIN			:=0;
   		HMI_RO_SD_FLUSHING_MIN		:=0;
   		HMI_RO_HIGH_PUMP_SHUTDOWN	:=0;
   		HMI_P5_SD_FLUSHING_DONE.ON	:=0;
   		HMI_MV501_TIMEOUT_TM		:=0;
   		HMI_MV502_TIMEOUT_TM		:=0;
   		HMI_MV503_TIMEOUT_TM		:=0;
   		HMI_MV504_TIMEOUT_TM		:=0;
   
   
   		IF NOT HMI_P_RO_HIGH_DUTY.Pump_Running OR _NEXT  THEN
   			_NEXT:=0;
   			HMI_P5_STATE:=15;
   		END_IF;
   
   	15:(*OPN MV504*)
   		_P_RO_HIGH_AutoInp	:= 0;
   		_MV501_AutoInp		:= 1;
   		_MV502_AutoInp		:= 1;
   		_MV503_AutoInp		:= 0;
   		_MV504_AutoInp		:= 1;
   
   		HMI_RO_HPP_SD.ON			:=0;
   		HMI_FLUSHING_MIN			:=0;
   		HMI_RO_SD_FLUSHING_MIN		:=0;
   		HMI_RO_HIGH_PUMP_SHUTDOWN	:=0;
   		HMI_P5_SD_FLUSHING_DONE.ON	:=0;
   		HMI_MV501_TIMEOUT_TM		:=0;
   		HMI_MV502_TIMEOUT_TM		:=0;
   		HMI_MV503_TIMEOUT_TM		:=0;
   	(*	HMI_MV504_TIMEOUT_TM		:=0;*)
   
   		IF _SEC_P THEN
   			HMI_MV504_TIMEOUT_TM:= HMI_MV504_TIMEOUT_TM+1;
   		END_IF;
   
   		IF HMI_MV504.STATUS=2 OR _NEXT OR HMI_MV504_TIMEOUT_TM >120 THEN
   			_NEXT:=0;
   			HMI_P5_STATE:=16;
   		END_IF;
   
   	16:(*CLOSE MV502*)
   		_P_RO_HIGH_AutoInp	:= 0;
   		_MV501_AutoInp		:= 1;
   		_MV502_AutoInp		:= 0;
   		_MV503_AutoInp		:= 0;
   		_MV504_AutoInp		:= 1;
   
   		HMI_RO_HPP_SD.ON			:=0;
   		HMI_FLUSHING_MIN			:=0;
   		HMI_RO_SD_FLUSHING_MIN		:=0;
   		HMI_RO_HIGH_PUMP_SHUTDOWN	:=0;
   		HMI_P5_SD_FLUSHING_DONE.ON	:=0;
   		HMI_MV501_TIMEOUT_TM		:=0;
   		(*HMI_MV502_TIMEOUT_TM		:=0;*)
   		HMI_MV503_TIMEOUT_TM		:=0;
   		HMI_MV504_TIMEOUT_TM		:=0;
   
   		IF _SEC_P THEN
   			HMI_MV502_TIMEOUT_TM:= HMI_MV502_TIMEOUT_TM+1;
   		END_IF;
   
   		IF HMI_MV502.STATUS=1 OR _NEXT OR HMI_MV502_TIMEOUT_TM >120 THEN
   			_NEXT:=0;
   			HMI_P5_STATE:=17;
   		END_IF;
   
   	17:(*OPEN MV503*)
   		_P_RO_HIGH_AutoInp	:= 0;
   		_MV501_AutoInp		:= 1;
   		_MV502_AutoInp		:= 0;
   		_MV503_AutoInp		:= 1;
   		_MV504_AutoInp		:= 1;
   
   		HMI_RO_HPP_SD.ON			:=0;
   		HMI_FLUSHING_MIN			:=0;
   		HMI_RO_SD_FLUSHING_MIN		:=0;
   		HMI_RO_HIGH_PUMP_SHUTDOWN	:=0;
   		HMI_P5_SD_FLUSHING_DONE.ON	:=0;
   		HMI_MV501_TIMEOUT_TM		:=0;
   		HMI_MV502_TIMEOUT_TM		:=0;
   		(*HMI_MV503_TIMEOUT_TM		:=0;*)
   		HMI_MV504_TIMEOUT_TM		:=0;
   
   		IF _SEC_P THEN
   			HMI_MV503_TIMEOUT_TM:= HMI_MV503_TIMEOUT_TM+1;
   		END_IF;
   
   
   		IF HMI_MV503.STATUS=2 OR _NEXT OR HMI_MV503_TIMEOUT_TM >120  THEN
   			_NEXT:=0;
   			HMI_P5_STATE:=18;
   		END_IF;
   
   	18:(*CLOSE MV501*)
   		_P_RO_HIGH_AutoInp	:= 0;
   		_MV501_AutoInp		:= 0;
   		_MV502_AutoInp		:= 0;
   		_MV503_AutoInp		:= 1;
   		_MV504_AutoInp		:= 1;
   
   		HMI_RO_HPP_SD.ON			:=0;
   		HMI_FLUSHING_MIN			:=0;
   		HMI_RO_SD_FLUSHING_MIN		:=0;
   		HMI_RO_HIGH_PUMP_SHUTDOWN	:=0;
   		HMI_P5_SD_FLUSHING_DONE.ON	:=0;
   		(*HMI_MV501_TIMEOUT_TM		:=0;*)
   		HMI_MV502_TIMEOUT_TM		:=0;
   		HMI_MV503_TIMEOUT_TM		:=0;
   		HMI_MV504_TIMEOUT_TM		:=0;
   
   		IF HMI_MV501.STATUS=1 OR _NEXT OR HMI_MV501_TIMEOUT_TM >120  THEN
   			_NEXT:=0;
   			HMI_P5_STATE:=19;
   		END_IF;
   
   	19:(*KEEP RO FEED PUMP RUNNING  *)
   		_P_RO_HIGH_AutoInp	:= 0;
   		_MV501_AutoInp		:= 0;
   		_MV502_AutoInp		:= 0;
   		_MV503_AutoInp		:= 1;
   		_MV504_AutoInp		:= 1;
   		_P50X_AutoSpeed		:= HMI_VSD_MIN_SPEED;
   
   		HMI_RO_HPP_SD.ON			:=0;
   		HMI_FLUSHING_MIN			:=0;
   
   		HMI_RO_HIGH_PUMP_SHUTDOWN	:=0;
   		HMI_P5_SD_FLUSHING_DONE.ON	:=0;
   		HMI_MV501_TIMEOUT_TM		:=0;
   		HMI_MV502_TIMEOUT_TM		:=0;
   		HMI_MV503_TIMEOUT_TM		:=0;
   		HMI_MV504_TIMEOUT_TM		:=0;
   
   		IF _MIN_P THEN
   			HMI_RO_SD_FLUSHING_MIN:=HMI_RO_SD_FLUSHING_MIN+1;
   		END_IF;
   
   		IF HMI_RO_SD_FLUSHING_MIN>HMI_RO_SD_FLUSHING_MIN_SP OR _NEXT THEN
   			_NEXT:=0;
   			HMI_P5_STATE:=20;
   		END_IF;
   
   	20:(*SHUTDOWN RO FEED PUMP *)
   		_P_RO_HIGH_AutoInp	:= 0;
   		_MV501_AutoInp		:= 0;
   		_MV502_AutoInp		:= 0;
   		_MV503_AutoInp		:= 1;
   		_MV504_AutoInp		:= 1;
   		_P50X_AutoSpeed		:= HMI_VSD_MIN_SPEED;
   
   		HMI_RO_HPP_SD.ON			:=1;
   		HMI_FLUSHING_MIN			:=0;
   		HMI_RO_SD_FLUSHING_MIN		:=0;
   		HMI_RO_HIGH_PUMP_SHUTDOWN	:=0;
   		HMI_P5_SD_FLUSHING_DONE.ON	:=0;
   		HMI_MV501_TIMEOUT_TM		:=0;
   		HMI_MV502_TIMEOUT_TM		:=0;
   		HMI_MV503_TIMEOUT_TM		:=0;
   		HMI_MV504_TIMEOUT_TM		:=0;
   
   		IF (NOT HMI_P_RO_FEED_DUTY.Pump_Running ) OR _NEXT THEN
   			_NEXT:=0;
   			HMI_P5_STATE:=21;
   		END_IF;
   
   	21:(*CLOSE MV503,MV504*)
   		_P_RO_HIGH_AutoInp	:= 0;
   		_MV501_AutoInp		:= 0;
   		_MV502_AutoInp		:= 0;
   		_MV503_AutoInp		:= 0;
   		_MV504_AutoInp		:= 0;
   		_P50X_AutoSpeed		:= HMI_VSD_MIN_SPEED;
   		HMI_RO_HPP_SD.ON:=0;
   
   		HMI_FLUSHING_MIN			:=0;
   		HMI_RO_SD_FLUSHING_MIN		:=0;
   		HMI_RO_HIGH_PUMP_SHUTDOWN	:=0;
   		HMI_P5_SD_FLUSHING_DONE.ON	:=0;
   		HMI_MV501_TIMEOUT_TM		:=0;
   		HMI_MV502_TIMEOUT_TM		:=0;
   		(*HMI_MV503_TIMEOUT_TM		:=0;*)
   		(*HMI_MV504_TIMEOUT_TM		:=0;*)
   
   		IF _SEC_P THEN
   			HMI_MV503_TIMEOUT_TM:= HMI_MV503_TIMEOUT_TM+1;
   			HMI_MV504_TIMEOUT_TM:= HMI_MV504_TIMEOUT_TM+1;
   		END_IF;
   
   
   
   
   		IF HMI_MV503.STATUS=1 AND HMI_MV504.STATUS=1 OR _NEXT OR HMI_MV503_TIMEOUT_TM >120 OR HMI_MV504_TIMEOUT_TM >120  THEN
   			_NEXT:=0;
   
   
   			HMI_P5_STATE:=1;
   		END_IF;
   ELSE
   	HMI_P5_STATE:=1;
   END_CASE;
   
   
   
   
   
   
   
   
   
   
   
   
   
   
   
   
   
   
   
   
END_ROUTINE

ROUTINE MainRoutine   (* ladder *)
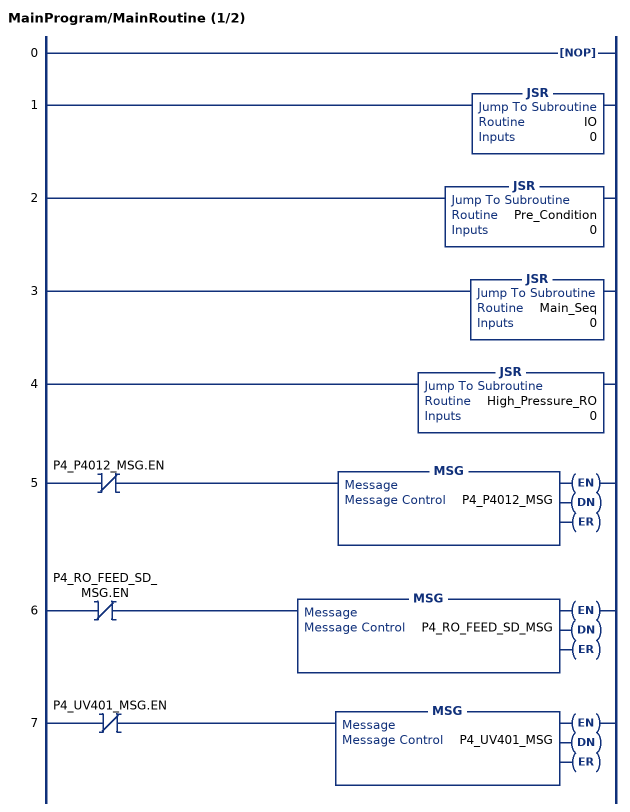
   0: NOP();
   1: JSR(IO,0);
   2: JSR(Pre_Condition,0);
   3: JSR(Main_Seq,0);
   4: JSR(High_Pressure_RO,0);
   5: XIO(P4_P4012_MSG.EN)MSG(P4_P4012_MSG);
   6: XIO(P4_RO_FEED_SD_MSG.EN)MSG(P4_RO_FEED_SD_MSG);
   7: XIO(P4_UV401_MSG.EN)MSG(P4_UV401_MSG);
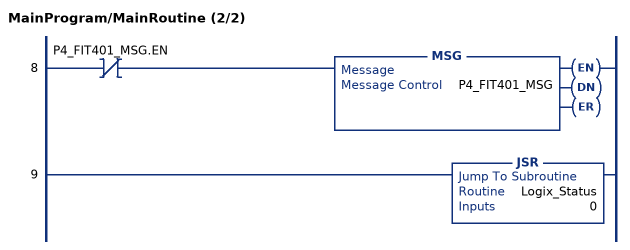
   8: XIO(P4_FIT401_MSG.EN)MSG(P4_FIT401_MSG);
   9: JSR(Logix_Status,0);
END_ROUTINE

ROUTINE Pre_Condition   (* structured text *)
   (*RESET ALL INSTRUMENT*)
   IF HMI_PLANT_RESET.ON THEN
   	HMI_P501.Reset	:=1;
   	HMI_P502.Reset	:=1;
   	HMI_MV501.Reset	:=1;
   	HMI_MV502.Reset	:=1;
   	HMI_MV503.Reset	:=1;
   	HMI_MV504.Reset :=1;
   
   END_IF;
   
   (*ALL INSTRUMENT IN AUTO MODE*)
   IF HMI_PLANT_AUTO.ON THEN
   	HMI_P501.Auto	:=1;
   	HMI_P502.Auto	:=1;
   	HMI_MV501.Auto	:=1;
   	HMI_MV502.Auto	:=1;
   	HMI_MV503.Auto	:=1;
   	HMI_MV504.Auto 	:=1;
   END_IF;
   
   (*ALL INSTRUMENT IN MANUAL MODE*)
   IF HMI_PLANT_AUTO.OFF THEN
   	HMI_P501.Auto	:=0;
   	HMI_P502.Auto	:=0;
   	HMI_MV501.Auto	:=0;
   	HMI_MV502.Auto	:=0;
   	HMI_MV503.Auto	:=0;
   	HMI_MV504.Auto 	:=0;
   END_IF;
   
   HMI_P5_PERMISSIVE.ON:= (HMI_P501.Avl OR HMI_P502.Avl) AND HMI_MV501.Avl AND HMI_MV502.Avl AND HMI_MV503.Avl AND HMI_MV504.Avl;
   
   
   (*Enable Flow Totalising*)
   _FIT501_Tot_Enb	:= HMI_P501.status=2 OR HMI_P502.status=2;
   _FIT502_Tot_Enb	:= HMI_MV501.status=2;
   _FIT503_Tot_Enb	:= HMI_P401.status=2 OR HMI_P402.status=2;
   _FIT504_Tot_Enb	:= HMI_P401.status=2 OR HMI_P402.status=2;
   
   TON_FIT401_TM.PRE 			:= 	3*1000;
   TON_FIT401_TM.TimerEnable 	:=  HMI_FIT401.ALL AND HMI_P_RO_FEED_DUTY.Pump_Running ;
   TONR(TON_FIT401_TM);
   
   (*P501 Permissive*)
   HMI_P501.Permissive.0 	:= HMI_P_RO_FEED_DUTY.Pump_Running;
   (*HMI_P501.Permissive.1 	:= NOT HMI_FIT401.ALL;
   HMI_P501.Permissive.2 	:= HMI_UV401.STATUS=2;*)
   HMI_P501.Permissive.1 	:= 1;
   HMI_P501.Permissive.2 	:= 1;
   HMI_P501.Permissive.3 	:= 1;
   HMI_P501.Permissive.4 	:= 1;
   HMI_P501.Permissive.5 	:= 1;
   HMI_P501.Permissive.6 	:= 1;
   HMI_P501.Permissive.7 	:= 1;
   HMI_P501.Permissive.8 	:= 1;
   HMI_P501.Permissive.9 	:= 1;
   HMI_P501.Permissive.10 	:= 1;
   HMI_P501.Permissive.11 	:= 1;
   HMI_P501.Permissive.12 	:= 1;
   HMI_P501.Permissive.13	:= 1;
   HMI_P501.Permissive.14	:= 1;
   HMI_P501.Permissive.15 	:= 1;
   
   HMI_P501_MSG.PERMISSIVE1 := HMI_P501.Permissive.0;
   HMI_P501_MSG.PERMISSIVE2 := HMI_P501.Permissive.1;
   HMI_P501_MSG.PERMISSIVE3 := HMI_P501.Permissive.2;
   HMI_P501_MSG.PERMISSIVE4 := 0;
   HMI_P501_MSG.PERMISSIVE5 := 0;
   
   (*P502 Permissive*)
   HMI_P502.Permissive.0 	:= HMI_P_RO_FEED_DUTY.Pump_Running;
   HMI_P502.Permissive.1 	:= NOT HMI_FIT401.ALL;
   HMI_P502.Permissive.2 	:= HMI_UV401.STATUS=2;
   HMI_P502.Permissive.3 	:= 1;
   HMI_P502.Permissive.4 	:= 1;
   HMI_P502.Permissive.5 	:= 1;
   HMI_P502.Permissive.6 	:= 1;
   HMI_P502.Permissive.7 	:= 1;
   HMI_P502.Permissive.8 	:= 1;
   HMI_P502.Permissive.9 	:= 1;
   HMI_P502.Permissive.10 	:= 1;
   HMI_P502.Permissive.11 	:= 1;
   HMI_P502.Permissive.12 	:= 1;
   HMI_P502.Permissive.13	:= 1;
   HMI_P502.Permissive.14	:= 1;
   HMI_P502.Permissive.15 	:= 1;
   
   HMI_P502_MSG.PERMISSIVE1 := HMI_P502.Permissive.0;
   HMI_P502_MSG.PERMISSIVE2 := HMI_P502.Permissive.1;
   HMI_P502_MSG.PERMISSIVE3 := HMI_P502.Permissive.2;
   HMI_P502_MSG.PERMISSIVE4 := 0;
   HMI_P502_MSG.PERMISSIVE5 := 0;
   
   (*-------------------------------------------------------------------------------------*)
   (*P501 Shutdown*)
   HMI_P501.SD.0 	:= NOT HMI_P_RO_FEED_DUTY.Pump_Running;
   (*HMI_P501.SD.1 	:= TON_FIT401_TM.DN;
   HMI_P501.SD.2 	:= HMI_UV401.STATUS<>2;*)
   HMI_P501.SD.1 := 0;
   HMI_P501.SD.2 := 0;
   HMI_P501.SD.3 	:= 0;(*HMI_PSL501.Alarm;*)
   HMI_P501.SD.4 	:= 0;(*HMI_PSH501.Alarm;*)
   HMI_P501.SD.5 	:= 0;
   HMI_P501.SD.6 	:= 0;
   HMI_P501.SD.7 	:= 0;
   HMI_P501.SD.8 	:= 0;
   HMI_P501.SD.9 	:= 0;
   HMI_P501.SD.10 	:= 0;
   HMI_P501.SD.11 	:= 0;
   HMI_P501.SD.12 	:= 0;
   HMI_P501.SD.13 	:= 0;
   HMI_P501.SD.14 	:= 0;
   HMI_P501.SD.15 	:= 0;
   
   HMI_P501_MSG.SHUTDOWN1 := HMI_P501.SHUTDOWN.0 ;
   HMI_P501_MSG.SHUTDOWN2 := HMI_P501.SHUTDOWN.1 ;
   HMI_P501_MSG.SHUTDOWN3 := HMI_P501.SHUTDOWN.2 ;
   HMI_P501_MSG.SHUTDOWN4 := HMI_P501.SHUTDOWN.3 ;
   HMI_P501_MSG.SHUTDOWN5 := HMI_P501.SHUTDOWN.4 ;
   
   (*P502 Shutdown*)
   HMI_P502.SD.0 	:= NOT HMI_P_RO_FEED_DUTY.Pump_Running;
   HMI_P502.SD.1 	:= TON_FIT401_TM.DN;
   HMI_P502.SD.2 	:= HMI_UV401.STATUS<>2;
   HMI_P502.SD.3 	:= 0;(*HMI_PSL501.Alarm;*)
   HMI_P502.SD.4 	:= 0;(*HMI_PSH501.Alarm;*)
   HMI_P502.SD.5 	:= 0;
   HMI_P502.SD.6 	:= 0;
   HMI_P502.SD.7 	:= 0;
   HMI_P502.SD.8 	:= 0;
   HMI_P502.SD.9 	:= 0;
   HMI_P502.SD.10 	:= 0;
   HMI_P502.SD.11 	:= 0;
   HMI_P502.SD.12 	:= 0;
   HMI_P502.SD.13 	:= 0;
   HMI_P502.SD.14 	:= 0;
   HMI_P502.SD.15 	:= 0;
   
   HMI_P502_MSG.SHUTDOWN1 := HMI_P502.SHUTDOWN.0 ;
   HMI_P502_MSG.SHUTDOWN2 := HMI_P502.SHUTDOWN.1 ;
   HMI_P502_MSG.SHUTDOWN3 := HMI_P502.SHUTDOWN.2 ;
   HMI_P502_MSG.SHUTDOWN4 := HMI_P502.SHUTDOWN.3 ;
   HMI_P502_MSG.SHUTDOWN5 := HMI_P502.SHUTDOWN.4 ;
END_ROUTINE
END_PROGRAM
